REGION Network 1: Conversion de temperatura leida por termopares a temperaturas para poder tratar en el codigo
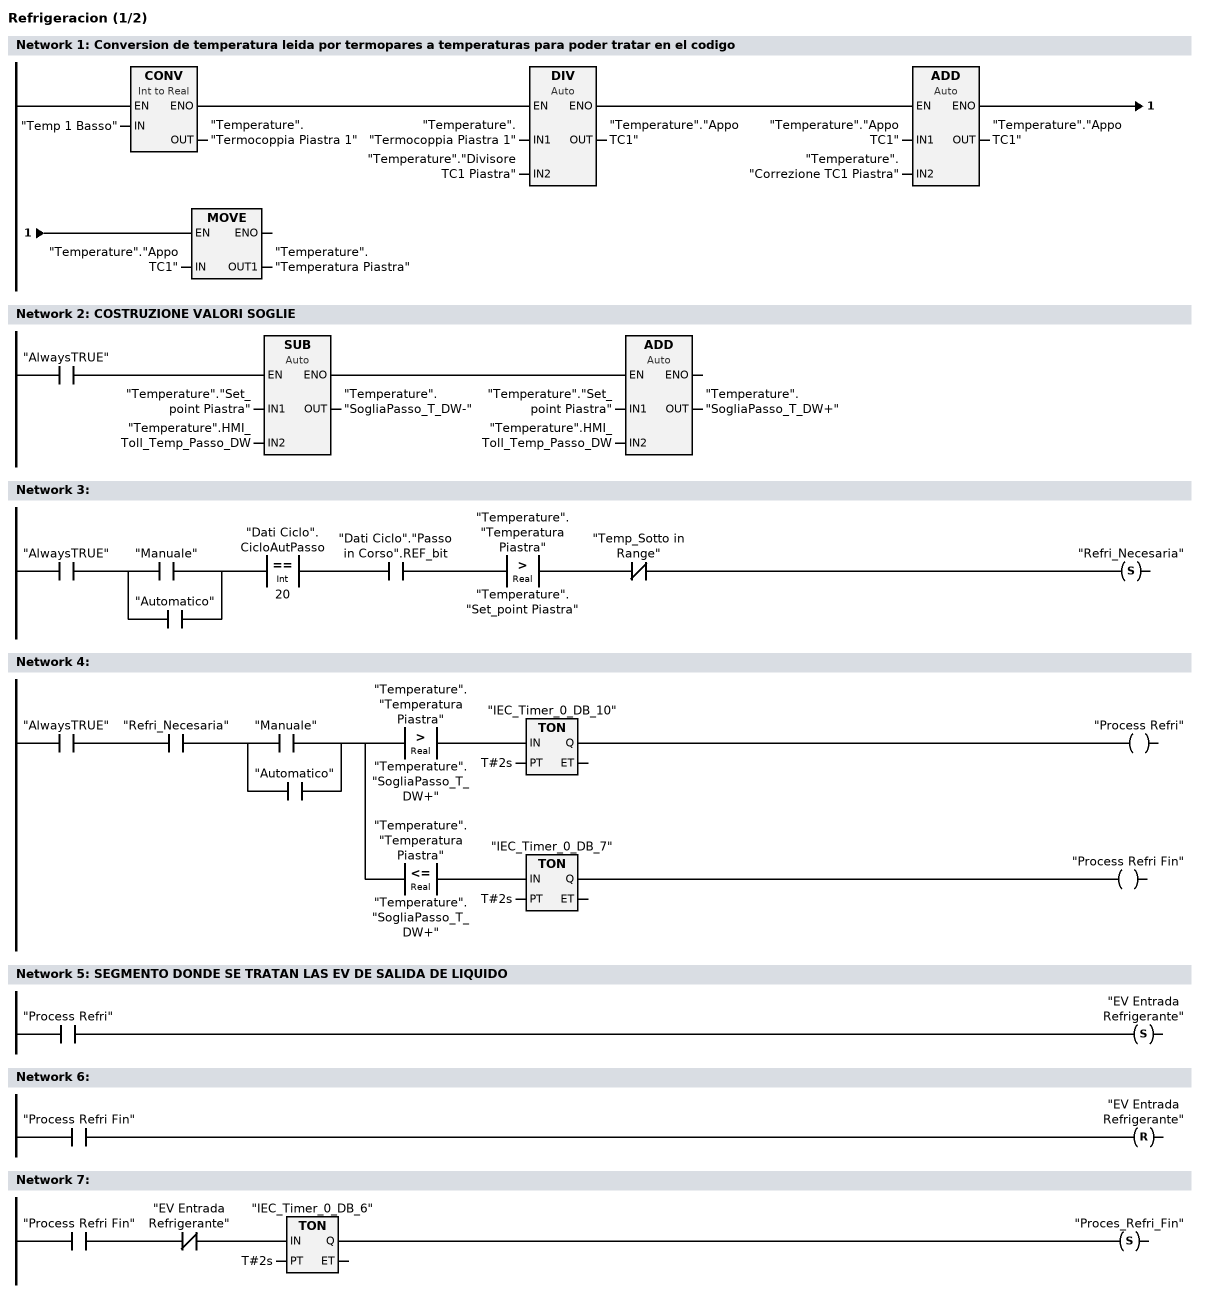
   RUNG wire#powerrail
      { S7_Templates := "[SrcType := Int, DestType := Real]" } Convert(in := "Temp 1 Basso", out => "Temperature"."Termocoppia Piastra 1")
      Div(in1 := "Temperature"."Termocoppia Piastra 1", in2 := "Temperature"."Divisore TC1 Piastra", out => "Temperature"."Appo TC1")
      Add(in1 := "Temperature"."Appo TC1", in2 := "Temperature"."Correzione TC1 Piastra", out => "Temperature"."Appo TC1")
      Move(in := "Temperature"."Appo TC1", out1 => "Temperature"."Temperatura Piastra")
   END_RUNG
   // the same network as SCL:
   "Temperature"."Termocoppia Piastra 1" := INT_TO_REAL("Temp 1 Basso");
   "Temperature"."Appo TC1" := "Temperature"."Termocoppia Piastra 1" / "Temperature"."Divisore TC1 Piastra";
   "Temperature"."Appo TC1" := "Temperature"."Appo TC1" + "Temperature"."Correzione TC1 Piastra";
   "Temperature"."Temperatura Piastra" := "Temperature"."Appo TC1";
END_REGION

REGION Network 2: COSTRUZIONE VALORI SOGLIE
   RUNG wire#powerrail
      Contact( "AlwaysTRUE" )
      Sub(in1 := "Temperature"."Set_point Piastra", in2 := "Temperature".HMI_Toll_Temp_Passo_DW, out => "Temperature"."SogliaPasso_T_DW-")
      Add(in1 := "Temperature"."Set_point Piastra", in2 := "Temperature".HMI_Toll_Temp_Passo_DW, out => "Temperature"."SogliaPasso_T_DW+")
   END_RUNG
   // the same network as SCL:
   IF "AlwaysTRUE" THEN
       "Temperature"."SogliaPasso_T_DW-" := "Temperature"."Set_point Piastra" - "Temperature".HMI_Toll_Temp_Passo_DW;
       "Temperature"."SogliaPasso_T_DW+" := "Temperature"."Set_point Piastra" + "Temperature".HMI_Toll_Temp_Passo_DW;
   END_IF;
END_REGION

REGION Network 3
   RUNG wire#powerrail
      Contact( "AlwaysTRUE" )
      wire#w1
      Contact( "Manuale" )
      wire#w2
      { S7_Templates := "SrcType := Int" } EQ_Contact(in1 := "Dati Ciclo".CicloAutPasso, in2 := 20)
      Contact( "Dati Ciclo"."Passo in Corso".REF_bit )
      { S7_Templates := "SrcType := Real" } GT_Contact(in1 := "Temperature"."Temperatura Piastra", in2 := "Temperature"."Set_point Piastra")
      I_Contact( "Temp_Sotto in Range" )
      S_Coil( "Refri_Necesaria" )
   END_RUNG
   RUNG wire#w1
      Contact( "Automatico" )
   END_RUNG wire#w2
   // the same network as SCL:
   IF "AlwaysTRUE" AND ("Manuale" OR "Automatico") AND ("Dati Ciclo".CicloAutPasso = 20) AND "Dati Ciclo"."Passo in Corso".REF_bit AND ("Temperature"."Temperatura Piastra" > "Temperature"."Set_point Piastra") AND NOT "Temp_Sotto in Range" THEN
       "Refri_Necesaria" := TRUE;
   END_IF;
END_REGION

REGION Network 4
   #_w1 := "AlwaysTRUE" AND "Refri_Necesaria" AND ("Manuale" OR "Automatico");
   "IEC_Timer_0_DB_10".TON(IN := #_w1 AND ("Temperature"."Temperatura Piastra" > "Temperature"."SogliaPasso_T_DW+"),
                           PT := T#2s);
   "Process Refri" := "IEC_Timer_0_DB_10".Q;
   "IEC_Timer_0_DB_7".TON(IN := #_w1 AND ("Temperature"."Temperatura Piastra" <= "Temperature"."SogliaPasso_T_DW+"),
                          PT := T#2s);
   "Process Refri Fin" := "IEC_Timer_0_DB_7".Q;
END_REGION

REGION Network 5: SEGMENTO DONDE SE TRATAN LAS EV DE SALIDA DE LIQUIDO
   RUNG wire#powerrail
      Contact( "Process Refri" )
      S_Coil( "EV Entrada Refrigerante" )
   END_RUNG
   // the same network as SCL:
   IF "Process Refri" THEN "EV Entrada Refrigerante" := TRUE; END_IF;
END_REGION

REGION Network 6
   RUNG wire#powerrail
      Contact( "Process Refri Fin" )
      R_Coil( "EV Entrada Refrigerante" )
   END_RUNG
   // the same network as SCL:
   IF "Process Refri Fin" THEN "EV Entrada Refrigerante" := FALSE; END_IF;
END_REGION

REGION Network 7
   "IEC_Timer_0_DB_6".TON(IN := "Process Refri Fin" AND NOT "EV Entrada Refrigerante", PT := T#2s);
   IF "IEC_Timer_0_DB_6".Q THEN "Proces_Refri_Fin" := TRUE; END_IF;
END_REGION

REGION Network 8
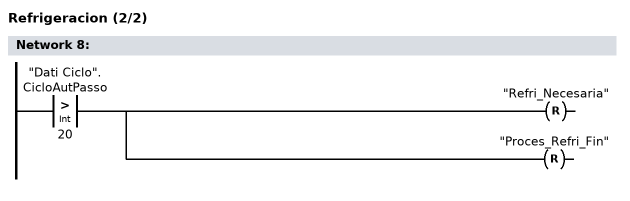
   RUNG wire#powerrail
      { S7_Templates := "SrcType := Int" } GT_Contact(in1 := "Dati Ciclo".CicloAutPasso, in2 := 20)
      wire#w1
      R_Coil( "Refri_Necesaria" )
   END_RUNG
   RUNG wire#w1
      R_Coil( "Proces_Refri_Fin" )
   END_RUNG
   // the same network as SCL:
   IF "Dati Ciclo".CicloAutPasso > 20 THEN
       "Refri_Necesaria" := FALSE;
       "Proces_Refri_Fin" := FALSE;
   END_IF;
END_REGION
END_FUNCTION

FUNCTION "Temperatura Sopra" : Void   // FC11, LAD
{ S7_Optimized_Access := 'TRUE' }
VERSION : 0.1
   VAR_TEMP   // added for the SCL form of the ladder/FBD networks
      _w1 : Bool;
   END_VAR
BEGIN

REGION Network 1: Costruzione valore temperatura
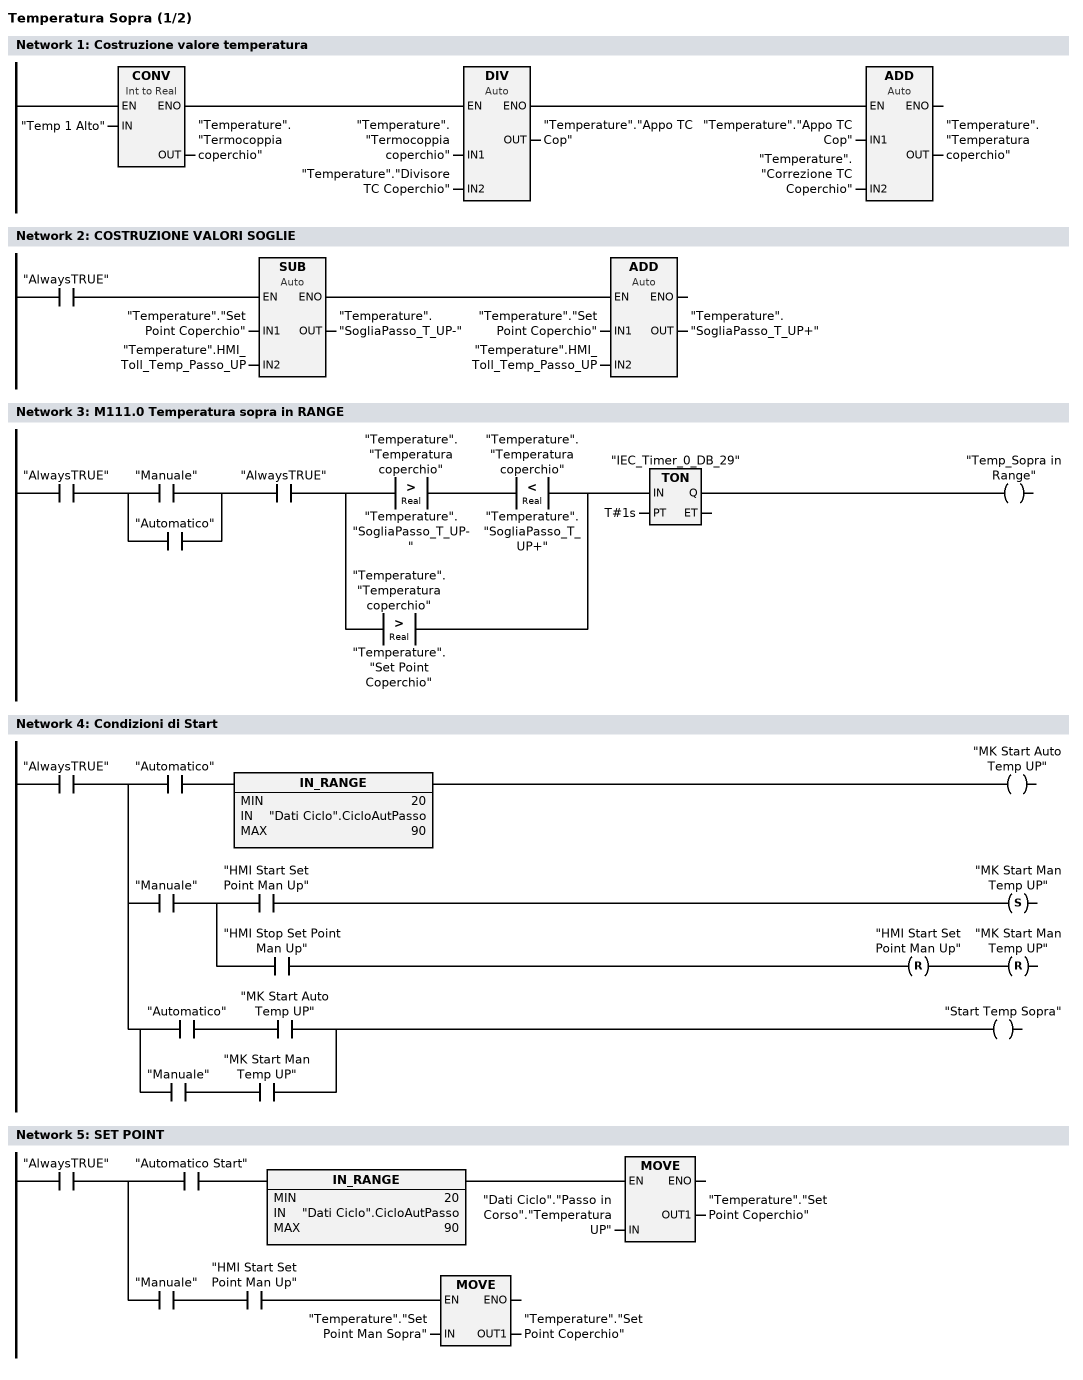
   RUNG wire#powerrail
      { S7_Templates := "[SrcType := Int, DestType := Real]" } Convert(in := "Temp 1 Alto", out => "Temperature"."Termocoppia coperchio")
      Div(in1 := "Temperature"."Termocoppia coperchio", in2 := "Temperature"."Divisore TC Coperchio", out => "Temperature"."Appo TC Cop")
      Add(in1 := "Temperature"."Appo TC Cop", in2 := "Temperature"."Correzione TC Coperchio", out => "Temperature"."Temperatura coperchio")
   END_RUNG
   // the same network as SCL:
   "Temperature"."Termocoppia coperchio" := INT_TO_REAL("Temp 1 Alto");
   "Temperature"."Appo TC Cop" := "Temperature"."Termocoppia coperchio" / "Temperature"."Divisore TC Coperchio";
   "Temperature"."Temperatura coperchio" := "Temperature"."Appo TC Cop" + "Temperature"."Correzione TC Coperchio";
END_REGION

REGION Network 2: COSTRUZIONE VALORI SOGLIE
   RUNG wire#powerrail
      Contact( "AlwaysTRUE" )
      Sub(in1 := "Temperature"."Set Point Coperchio", in2 := "Temperature".HMI_Toll_Temp_Passo_UP, out => "Temperature"."SogliaPasso_T_UP-")
      Add(in1 := "Temperature"."Set Point Coperchio", in2 := "Temperature".HMI_Toll_Temp_Passo_UP, out => "Temperature"."SogliaPasso_T_UP+")
   END_RUNG
   // the same network as SCL:
   IF "AlwaysTRUE" THEN
       "Temperature"."SogliaPasso_T_UP-" := "Temperature"."Set Point Coperchio" - "Temperature".HMI_Toll_Temp_Passo_UP;
       "Temperature"."SogliaPasso_T_UP+" := "Temperature"."Set Point Coperchio" + "Temperature".HMI_Toll_Temp_Passo_UP;
   END_IF;
END_REGION

REGION Network 3: M111.0 Temperatura sopra in RANGE
   "IEC_Timer_0_DB_29".TON(IN := "AlwaysTRUE" AND ("Manuale" OR "Automatico") AND "AlwaysTRUE" AND ((("Temperature"."Temperatura coperchio" > "Temperature"."SogliaPasso_T_UP-") AND ("Temperature"."Temperatura coperchio" < "Temperature"."SogliaPasso_T_UP+")) OR ("Temperature"."Temperatura coperchio" > "Temperature"."Set Point Coperchio")),
                           PT := T#1s);
   "Temp_Sopra in Range" := "IEC_Timer_0_DB_29".Q;
END_REGION

REGION Network 4: Condizioni di Start
   RUNG wire#powerrail
      Contact( "AlwaysTRUE" )
      wire#w1
      Contact( "Automatico" )
      { S7_Templates := "SrcType := Int" } InRange(min := 20, in := "Dati Ciclo".CicloAutPasso, max := 90)
      Coil( "MK Start Auto Temp UP" )
   END_RUNG
   RUNG wire#w1
      Contact( "Manuale" )
      wire#w2
      Contact( "HMI Start Set Point Man Up" )
      S_Coil( "MK Start Man Temp UP" )
   END_RUNG
   RUNG wire#w2
      Contact( "HMI Stop Set Point Man Up" )
      R_Coil( "HMI Start Set Point Man Up" )
      R_Coil( "MK Start Man Temp UP" )
   END_RUNG
   RUNG wire#w1
      Contact( "Automatico" )
      Contact( "MK Start Auto Temp UP" )
      wire#w3
      Coil( "Start Temp Sopra" )
   END_RUNG
   RUNG wire#w1
      Contact( "Manuale" )
      Contact( "MK Start Man Temp UP" )
   END_RUNG wire#w3
   // the same network as SCL:
   "MK Start Auto Temp UP" := "AlwaysTRUE" AND "Automatico" AND (20 <= "Dati Ciclo".CicloAutPasso) AND ("Dati Ciclo".CicloAutPasso <= 90);
   #_w1 := "AlwaysTRUE" AND "Manuale";
   IF #_w1 AND "HMI Start Set Point Man Up" THEN "MK Start Man Temp UP" := TRUE; END_IF;
   IF #_w1 AND "HMI Stop Set Point Man Up" THEN
       "HMI Start Set Point Man Up" := FALSE;
       "MK Start Man Temp UP" := FALSE;
   END_IF;
   "Start Temp Sopra" := "AlwaysTRUE" AND (("Automatico" AND "MK Start Auto Temp UP") OR ("Manuale" AND "MK Start Man Temp UP"));
END_REGION

REGION Network 5: SET POINT
   RUNG wire#powerrail
      Contact( "AlwaysTRUE" )
      wire#w1
      Contact( "Automatico Start" )
      { S7_Templates := "SrcType := Int" } InRange(min := 20, in := "Dati Ciclo".CicloAutPasso, max := 90)
      Move(in := "Dati Ciclo"."Passo in Corso"."Temperatura UP", out1 => "Temperature"."Set Point Coperchio")
   END_RUNG
   RUNG wire#w1
      Contact( "Manuale" )
      Contact( "HMI Start Set Point Man Up" )
      Move(in := "Temperature"."Set Point Man Sopra", out1 => "Temperature"."Set Point Coperchio")
   END_RUNG
   // the same network as SCL:
   IF "AlwaysTRUE" AND "Automatico Start" AND (20 <= "Dati Ciclo".CicloAutPasso) AND ("Dati Ciclo".CicloAutPasso <= 90) THEN
       "Temperature"."Set Point Coperchio" := "Dati Ciclo"."Passo in Corso"."Temperatura UP";
   END_IF;
   IF "AlwaysTRUE" AND "Manuale" AND "HMI Start Set Point Man Up" THEN
       "Temperature"."Set Point Coperchio" := "Temperature"."Set Point Man Sopra";
   END_IF;
END_REGION

REGION Network 6: Comando resistenze
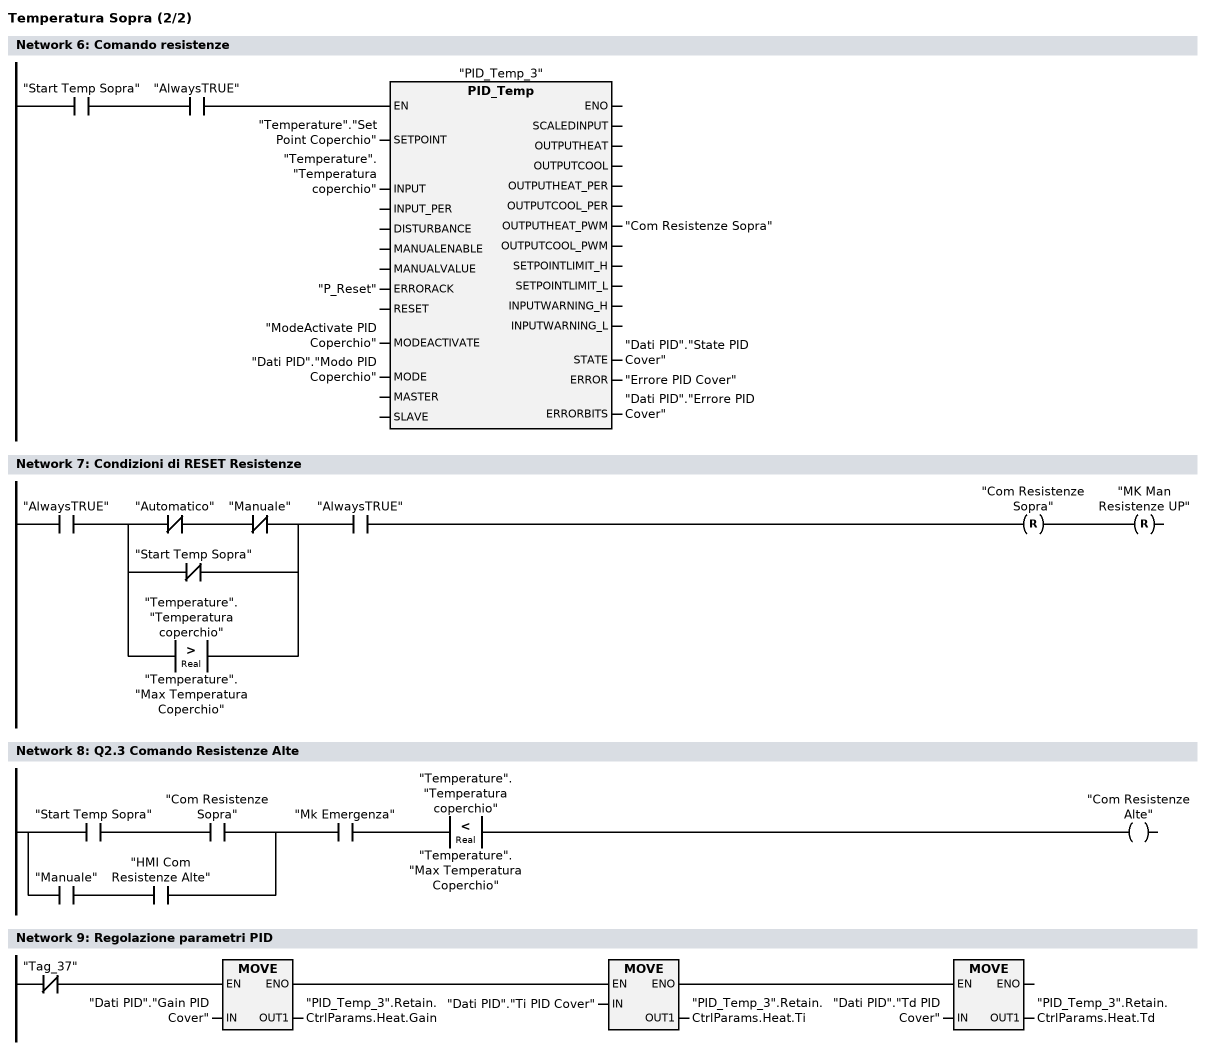
   IF "Start Temp Sopra" AND "AlwaysTRUE" THEN
       "PID_Temp_3"(Setpoint := "Temperature"."Set Point Coperchio",   // PID_Temp
                    Input := "Temperature"."Temperatura coperchio",
                    ErrorAck := "P_Reset",
                    ModeActivate := "ModeActivate PID Coperchio",
                    Mode := "Dati PID"."Modo PID Coperchio",
                    OutputHeat_PWM => "Com Resistenze Sopra",
                    State => "Dati PID"."State PID Cover",
                    Error => "Errore PID Cover",
                    ErrorBits => "Dati PID"."Errore PID Cover");
   END_IF;
END_REGION

REGION Network 7: Condizioni di RESET Resistenze
   RUNG wire#powerrail
      Contact( "AlwaysTRUE" )
      wire#w1
      I_Contact( "Automatico" )
      I_Contact( "Manuale" )
      wire#w2
      Contact( "AlwaysTRUE" )
      R_Coil( "Com Resistenze Sopra" )
      R_Coil( "MK Man Resistenze UP" )
   END_RUNG
   RUNG wire#w1
      I_Contact( "Start Temp Sopra" )
   END_RUNG wire#w2
   RUNG wire#w1
      { S7_Templates := "SrcType := Real" } GT_Contact(in1 := "Temperature"."Temperatura coperchio", in2 := "Temperature"."Max Temperatura Coperchio")
   END_RUNG wire#w2
   // the same network as SCL:
   IF "AlwaysTRUE" AND ((NOT "Automatico" AND NOT "Manuale") OR NOT "Start Temp Sopra" OR ("Temperature"."Temperatura coperchio" > "Temperature"."Max Temperatura Coperchio")) AND "AlwaysTRUE" THEN
       "Com Resistenze Sopra" := FALSE;
       "MK Man Resistenze UP" := FALSE;
   END_IF;
END_REGION

REGION Network 8: Q2.3 Comando Resistenze Alte
   RUNG wire#powerrail
      Contact( "Start Temp Sopra" )
      Contact( "Com Resistenze Sopra" )
      wire#w1
      Contact( "Mk Emergenza" )
      { S7_Templates := "SrcType := Real" } LT_Contact(in1 := "Temperature"."Temperatura coperchio", in2 := "Temperature"."Max Temperatura Coperchio")
      Coil( "Com Resistenze Alte" )
   END_RUNG
   RUNG wire#powerrail
      Contact( "Manuale" )
      Contact( "HMI Com Resistenze Alte" )
   END_RUNG wire#w1
   // the same network as SCL:
   "Com Resistenze Alte" := (("Start Temp Sopra" AND "Com Resistenze Sopra") OR ("Manuale" AND "HMI Com Resistenze Alte")) AND "Mk Emergenza" AND ("Temperature"."Temperatura coperchio" < "Temperature"."Max Temperatura Coperchio");
END_REGION

REGION Network 9: Regolazione parametri PID
   RUNG wire#powerrail
      I_Contact( "Tag_37" )
      Move(in := "Dati PID"."Gain PID Cover", out1 => "PID_Temp_3".Retain.CtrlParams.Heat.Gain)
      Move(in := "Dati PID"."Ti PID Cover", out1 => "PID_Temp_3".Retain.CtrlParams.Heat.Ti)
      Move(in := "Dati PID"."Td PID Cover", out1 => "PID_Temp_3".Retain.CtrlParams.Heat.Td)
   END_RUNG
   // the same network as SCL:
   IF NOT "Tag_37" THEN
       "PID_Temp_3".Retain.CtrlParams.Heat.Gain := "Dati PID"."Gain PID Cover";
       "PID_Temp_3".Retain.CtrlParams.Heat.Ti := "Dati PID"."Ti PID Cover";
       "PID_Temp_3".Retain.CtrlParams.Heat.Td := "Dati PID"."Td PID Cover";
   END_IF;
END_REGION
END_FUNCTION

FUNCTION "Vuoto Sotto" : Void   // FC12, LAD
{ S7_Optimized_Access := 'TRUE' }
VERSION : 0.1
   VAR_TEMP   // added for the SCL form of the ladder/FBD networks
      _w1 : Bool;
      _w2 : Bool;
   END_VAR
BEGIN

REGION Network 1: Costruzione valore vuoto
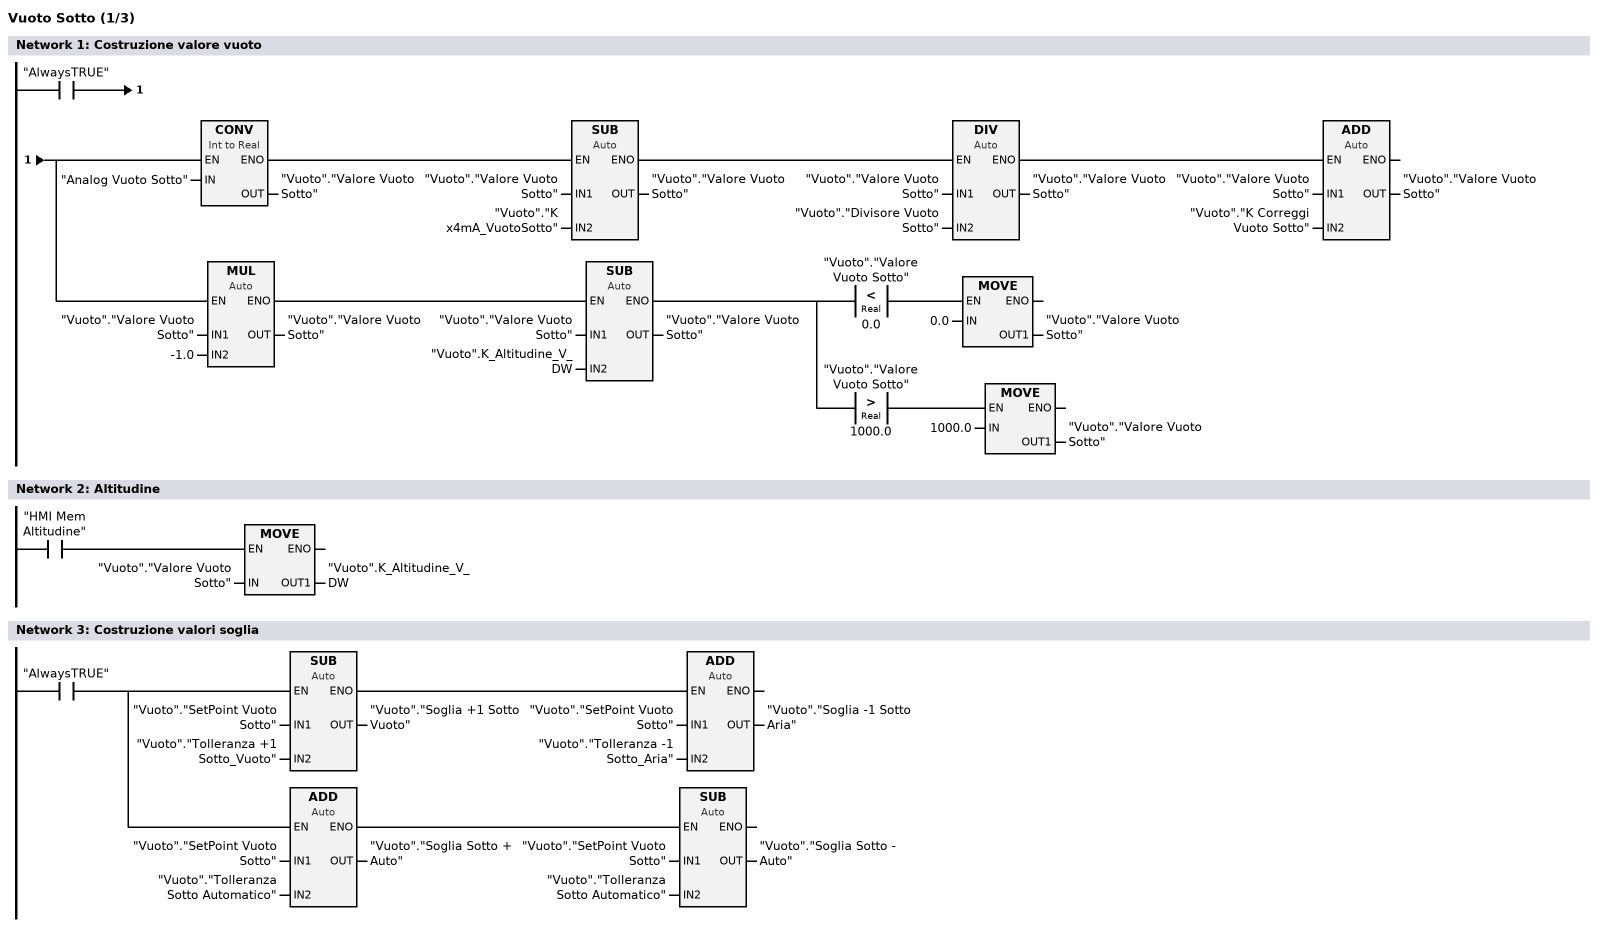
   RUNG wire#powerrail
      Contact( "AlwaysTRUE" )
      wire#w1
      { S7_Templates := "[SrcType := Int, DestType := Real]" } Convert(in := "Analog Vuoto Sotto", out => "Vuoto"."Valore Vuoto Sotto")
      Sub(in1 := "Vuoto"."Valore Vuoto Sotto", in2 := "Vuoto"."K x4mA_VuotoSotto", out => "Vuoto"."Valore Vuoto Sotto")
      Div(in1 := "Vuoto"."Valore Vuoto Sotto", in2 := "Vuoto"."Divisore Vuoto Sotto", out => "Vuoto"."Valore Vuoto Sotto")
      Add(in1 := "Vuoto"."Valore Vuoto Sotto", in2 := "Vuoto"."K Correggi Vuoto Sotto", out => "Vuoto"."Valore Vuoto Sotto")
   END_RUNG
   RUNG wire#w1
      Mul(in1 := "Vuoto"."Valore Vuoto Sotto", in2 := -1.0, out => "Vuoto"."Valore Vuoto Sotto")
      Sub(in1 := "Vuoto"."Valore Vuoto Sotto", in2 := "Vuoto".K_Altitudine_V_DW, out => "Vuoto"."Valore Vuoto Sotto")
      wire#w2
      { S7_Templates := "SrcType := Real" } LT_Contact(in1 := "Vuoto"."Valore Vuoto Sotto", in2 := 0.0)
      Move(in := 0.0, out1 => "Vuoto"."Valore Vuoto Sotto")
   END_RUNG
   RUNG wire#w2
      { S7_Templates := "SrcType := Real" } GT_Contact(in1 := "Vuoto"."Valore Vuoto Sotto", in2 := 1000.0)
      Move(in := 1000.0, out1 => "Vuoto"."Valore Vuoto Sotto")
   END_RUNG
   // the same network as SCL:
   IF "AlwaysTRUE" THEN
       "Vuoto"."Valore Vuoto Sotto" := INT_TO_REAL("Analog Vuoto Sotto");
       "Vuoto"."Valore Vuoto Sotto" := "Vuoto"."Valore Vuoto Sotto" - "Vuoto"."K x4mA_VuotoSotto";
       "Vuoto"."Valore Vuoto Sotto" := "Vuoto"."Valore Vuoto Sotto" / "Vuoto"."Divisore Vuoto Sotto";
       "Vuoto"."Valore Vuoto Sotto" := "Vuoto"."Valore Vuoto Sotto" + "Vuoto"."K Correggi Vuoto Sotto";
       "Vuoto"."Valore Vuoto Sotto" := "Vuoto"."Valore Vuoto Sotto" * (-1.0);
       "Vuoto"."Valore Vuoto Sotto" := "Vuoto"."Valore Vuoto Sotto" - "Vuoto".K_Altitudine_V_DW;
   END_IF;
   IF "AlwaysTRUE" AND ("Vuoto"."Valore Vuoto Sotto" < 0.0) THEN "Vuoto"."Valore Vuoto Sotto" := 0.0; END_IF;
   IF "AlwaysTRUE" AND ("Vuoto"."Valore Vuoto Sotto" > 1000.0) THEN
       "Vuoto"."Valore Vuoto Sotto" := 1000.0;
   END_IF;
END_REGION

REGION Network 2: Altitudine
   RUNG wire#powerrail
      Contact( "HMI Mem Altitudine" )
      Move(in := "Vuoto"."Valore Vuoto Sotto", out1 => "Vuoto".K_Altitudine_V_DW)
   END_RUNG
   // the same network as SCL:
   IF "HMI Mem Altitudine" THEN "Vuoto".K_Altitudine_V_DW := "Vuoto"."Valore Vuoto Sotto"; END_IF;
END_REGION

REGION Network 3: Costruzione valori soglia
   RUNG wire#powerrail
      Contact( "AlwaysTRUE" )
      wire#w1
      Sub(in1 := "Vuoto"."SetPoint Vuoto Sotto", in2 := "Vuoto"."Tolleranza +1 Sotto_Vuoto", out => "Vuoto"."Soglia +1 Sotto Vuoto")
      Add(in1 := "Vuoto"."SetPoint Vuoto Sotto", in2 := "Vuoto"."Tolleranza -1 Sotto_Aria", out => "Vuoto"."Soglia -1 Sotto Aria")
   END_RUNG
   RUNG wire#w1
      Add(in1 := "Vuoto"."SetPoint Vuoto Sotto", in2 := "Vuoto"."Tolleranza Sotto Automatico", out => "Vuoto"."Soglia Sotto + Auto")
      Sub(in1 := "Vuoto"."SetPoint Vuoto Sotto", in2 := "Vuoto"."Tolleranza Sotto Automatico", out => "Vuoto"."Soglia Sotto - Auto")
   END_RUNG
   // the same network as SCL:
   IF "AlwaysTRUE" THEN
       "Vuoto"."Soglia +1 Sotto Vuoto" := "Vuoto"."SetPoint Vuoto Sotto" - "Vuoto"."Tolleranza +1 Sotto_Vuoto";
       "Vuoto"."Soglia -1 Sotto Aria" := "Vuoto"."SetPoint Vuoto Sotto" + "Vuoto"."Tolleranza -1 Sotto_Aria";
       "Vuoto"."Soglia Sotto + Auto" := "Vuoto"."SetPoint Vuoto Sotto" + "Vuoto"."Tolleranza Sotto Automatico";
       "Vuoto"."Soglia Sotto - Auto" := "Vuoto"."SetPoint Vuoto Sotto" - "Vuoto"."Tolleranza Sotto Automatico";
   END_IF;
END_REGION

REGION Network 4: Condizioni di start
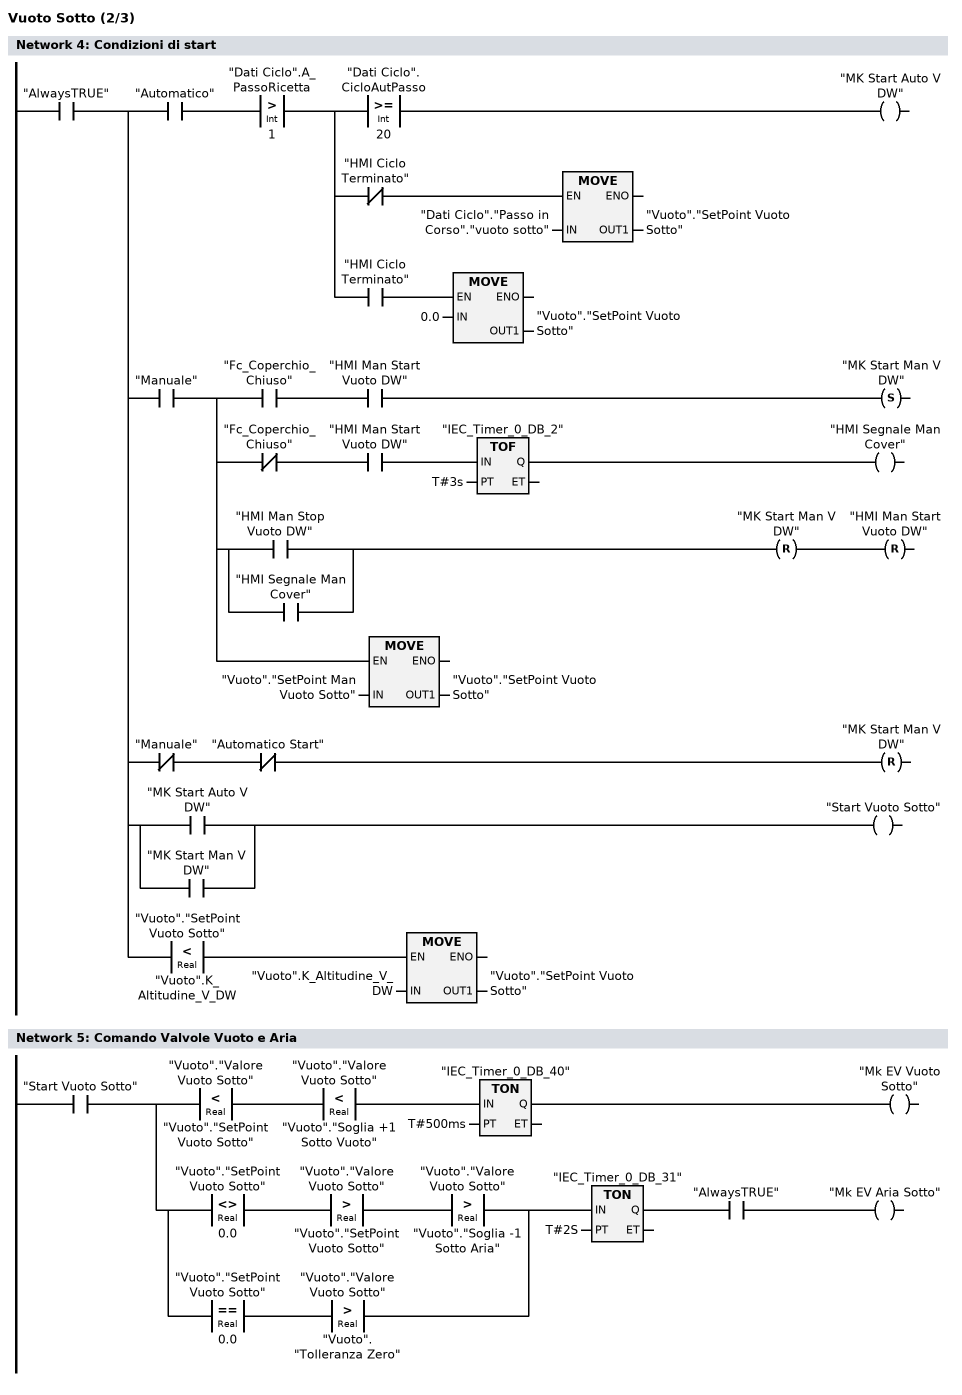
   #_w1 := "AlwaysTRUE" AND "Automatico" AND ("Dati Ciclo".A_PassoRicetta > 1);
   "MK Start Auto V DW" := #_w1 AND ("Dati Ciclo".CicloAutPasso >= 20);
   IF #_w1 AND NOT "HMI Ciclo Terminato" THEN
       "Vuoto"."SetPoint Vuoto Sotto" := "Dati Ciclo"."Passo in Corso"."vuoto sotto";
   END_IF;
   IF #_w1 AND "HMI Ciclo Terminato" THEN "Vuoto"."SetPoint Vuoto Sotto" := 0.0; END_IF;
   #_w2 := "AlwaysTRUE" AND "Manuale";
   IF #_w2 AND "Fc_Coperchio_Chiuso" AND "HMI Man Start Vuoto DW" THEN "MK Start Man V DW" := TRUE; END_IF;
   "IEC_Timer_0_DB_2".TOF(IN := #_w2 AND NOT "Fc_Coperchio_Chiuso" AND "HMI Man Start Vuoto DW", PT := T#3s);
   "HMI Segnale Man Cover" := "IEC_Timer_0_DB_2".Q;
   IF #_w2 AND ("HMI Man Stop Vuoto DW" OR "HMI Segnale Man Cover") THEN
       "MK Start Man V DW" := FALSE;
       "HMI Man Start Vuoto DW" := FALSE;
   END_IF;
   IF #_w2 THEN "Vuoto"."SetPoint Vuoto Sotto" := "Vuoto"."SetPoint Man Vuoto Sotto"; END_IF;
   IF "AlwaysTRUE" AND NOT "Manuale" AND NOT "Automatico Start" THEN "MK Start Man V DW" := FALSE; END_IF;
   "Start Vuoto Sotto" := "AlwaysTRUE" AND ("MK Start Auto V DW" OR "MK Start Man V DW");
   IF "AlwaysTRUE" AND ("Vuoto"."SetPoint Vuoto Sotto" < "Vuoto".K_Altitudine_V_DW) THEN
       "Vuoto"."SetPoint Vuoto Sotto" := "Vuoto".K_Altitudine_V_DW;
   END_IF;
END_REGION

REGION Network 5: Comando Valvole Vuoto e Aria
   "IEC_Timer_0_DB_40".TON(IN := "Start Vuoto Sotto" AND ("Vuoto"."Valore Vuoto Sotto" < "Vuoto"."SetPoint Vuoto Sotto") AND ("Vuoto"."Valore Vuoto Sotto" < "Vuoto"."Soglia +1 Sotto Vuoto"),
                           PT := T#500ms);
   "Mk EV Vuoto Sotto" := "IEC_Timer_0_DB_40".Q;
   "IEC_Timer_0_DB_31".TON(IN := "Start Vuoto Sotto" AND ((("Vuoto"."SetPoint Vuoto Sotto" <> 0.0) AND ("Vuoto"."Valore Vuoto Sotto" > "Vuoto"."SetPoint Vuoto Sotto") AND ("Vuoto"."Valore Vuoto Sotto" > "Vuoto"."Soglia -1 Sotto Aria")) OR (("Vuoto"."SetPoint Vuoto Sotto" = 0.0) AND ("Vuoto"."Valore Vuoto Sotto" > "Vuoto"."Tolleranza Zero"))),
                           PT := T#2S);
   "Mk EV Aria Sotto" := "IEC_Timer_0_DB_31".Q AND "AlwaysTRUE";
END_REGION

REGION Network 6: Vuoto in Range
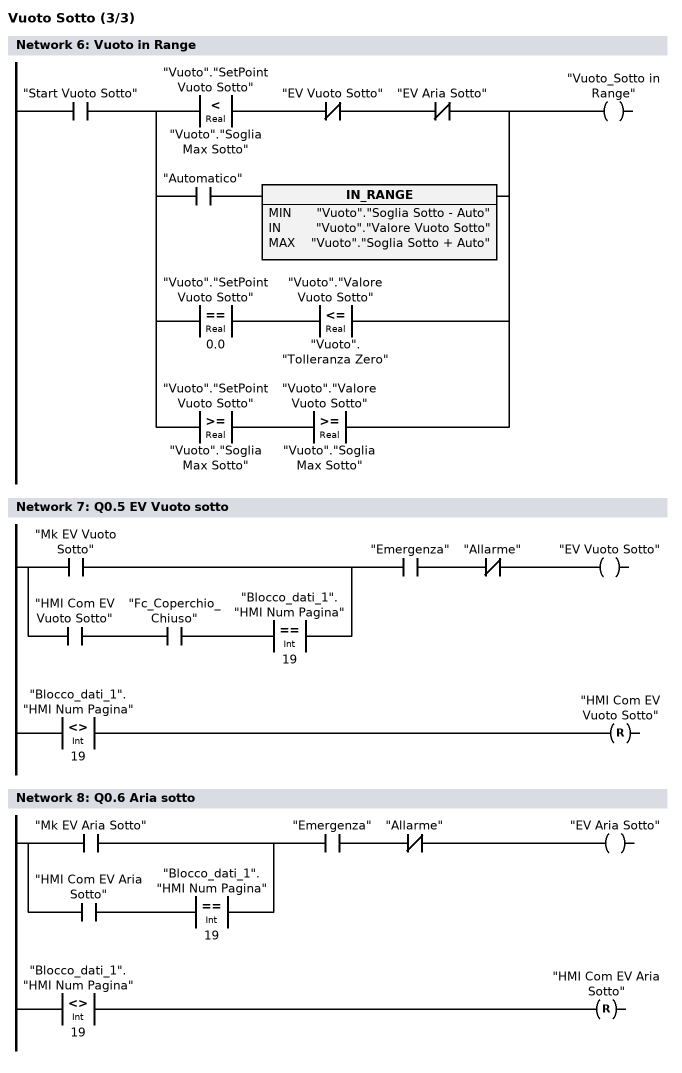
   RUNG wire#powerrail
      Contact( "Start Vuoto Sotto" )
      wire#w1
      { S7_Templates := "SrcType := Real" } LT_Contact(in1 := "Vuoto"."SetPoint Vuoto Sotto", in2 := "Vuoto"."Soglia Max Sotto")
      I_Contact( "EV Vuoto Sotto" )
      I_Contact( "EV Aria Sotto" )
      wire#w2
      Coil( "Vuoto_Sotto in Range" )
   END_RUNG
   RUNG wire#w1
      Contact( "Automatico" )
      { S7_Templates := "SrcType := Real" } InRange(min := "Vuoto"."Soglia Sotto - Auto", in := "Vuoto"."Valore Vuoto Sotto", max := "Vuoto"."Soglia Sotto + Auto")
   END_RUNG wire#w2
   RUNG wire#w1
      { S7_Templates := "SrcType := Real" } EQ_Contact(in1 := "Vuoto"."SetPoint Vuoto Sotto", in2 := 0.0)
      { S7_Templates := "SrcType := Real" } LE_Contact(in1 := "Vuoto"."Valore Vuoto Sotto", in2 := "Vuoto"."Tolleranza Zero")
   END_RUNG wire#w2
   RUNG wire#w1
      { S7_Templates := "SrcType := Real" } GE_Contact(in1 := "Vuoto"."SetPoint Vuoto Sotto", in2 := "Vuoto"."Soglia Max Sotto")
      { S7_Templates := "SrcType := Real" } GE_Contact(in1 := "Vuoto"."Valore Vuoto Sotto", in2 := "Vuoto"."Soglia Max Sotto")
   END_RUNG wire#w2
   // the same network as SCL:
   "Vuoto_Sotto in Range" := "Start Vuoto Sotto" AND ((("Vuoto"."SetPoint Vuoto Sotto" < "Vuoto"."Soglia Max Sotto") AND NOT "EV Vuoto Sotto" AND NOT "EV Aria Sotto") OR ("Automatico" AND ("Vuoto"."Soglia Sotto - Auto" <= "Vuoto"."Valore Vuoto Sotto") AND ("Vuoto"."Valore Vuoto Sotto" <= "Vuoto"."Soglia Sotto + Auto")) OR (("Vuoto"."SetPoint Vuoto Sotto" = 0.0) AND ("Vuoto"."Valore Vuoto Sotto" <= "Vuoto"."Tolleranza Zero")) OR (("Vuoto"."SetPoint Vuoto Sotto" >= "Vuoto"."Soglia Max Sotto") AND ("Vuoto"."Valore Vuoto Sotto" >= "Vuoto"."Soglia Max Sotto")));
END_REGION

REGION Network 7: Q0.5 EV Vuoto sotto
   RUNG wire#powerrail
      Contact( "Mk EV Vuoto Sotto" )
      wire#w1
      Contact( "Emergenza" )
      I_Contact( "Allarme" )
      Coil( "EV Vuoto Sotto" )
   END_RUNG
   RUNG wire#powerrail
      Contact( "HMI Com EV Vuoto Sotto" )
      Contact( "Fc_Coperchio_Chiuso" )
      { S7_Templates := "SrcType := Int" } EQ_Contact(in1 := "Blocco_dati_1"."HMI Num Pagina", in2 := 19)
   END_RUNG wire#w1
   RUNG wire#powerrail
      { S7_Templates := "SrcType := Int" } NE_Contact(in1 := "Blocco_dati_1"."HMI Num Pagina", in2 := 19)
      R_Coil( "HMI Com EV Vuoto Sotto" )
   END_RUNG
   // the same network as SCL:
   "EV Vuoto Sotto" := ("Mk EV Vuoto Sotto" OR ("HMI Com EV Vuoto Sotto" AND "Fc_Coperchio_Chiuso" AND ("Blocco_dati_1"."HMI Num Pagina" = 19))) AND "Emergenza" AND NOT "Allarme";
   IF "Blocco_dati_1"."HMI Num Pagina" <> 19 THEN "HMI Com EV Vuoto Sotto" := FALSE; END_IF;
END_REGION

REGION Network 8: Q0.6 Aria sotto
   RUNG wire#powerrail
      Contact( "Mk EV Aria Sotto" )
      wire#w1
      Contact( "Emergenza" )
      I_Contact( "Allarme" )
      Coil( "EV Aria Sotto" )
   END_RUNG
   RUNG wire#powerrail
      Contact( "HMI Com EV Aria Sotto" )
      { S7_Templates := "SrcType := Int" } EQ_Contact(in1 := "Blocco_dati_1"."HMI Num Pagina", in2 := 19)
   END_RUNG wire#w1
   RUNG wire#powerrail
      { S7_Templates := "SrcType := Int" } NE_Contact(in1 := "Blocco_dati_1"."HMI Num Pagina", in2 := 19)
      R_Coil( "HMI Com EV Aria Sotto" )
   END_RUNG
   // the same network as SCL:
   "EV Aria Sotto" := ("Mk EV Aria Sotto" OR ("HMI Com EV Aria Sotto" AND ("Blocco_dati_1"."HMI Num Pagina" = 19))) AND "Emergenza" AND NOT "Allarme";
   IF "Blocco_dati_1"."HMI Num Pagina" <> 19 THEN "HMI Com EV Aria Sotto" := FALSE; END_IF;
END_REGION
END_FUNCTION

FUNCTION "Vuoto Sopra" : Void   // FC13, LAD
{ S7_Optimized_Access := 'TRUE' }
VERSION : 0.1
   VAR_TEMP   // added for the SCL form of the ladder/FBD networks
      _w1 : Bool;
      _w2 : Bool;
   END_VAR
BEGIN

REGION Network 1: Costruzione valore vuoto
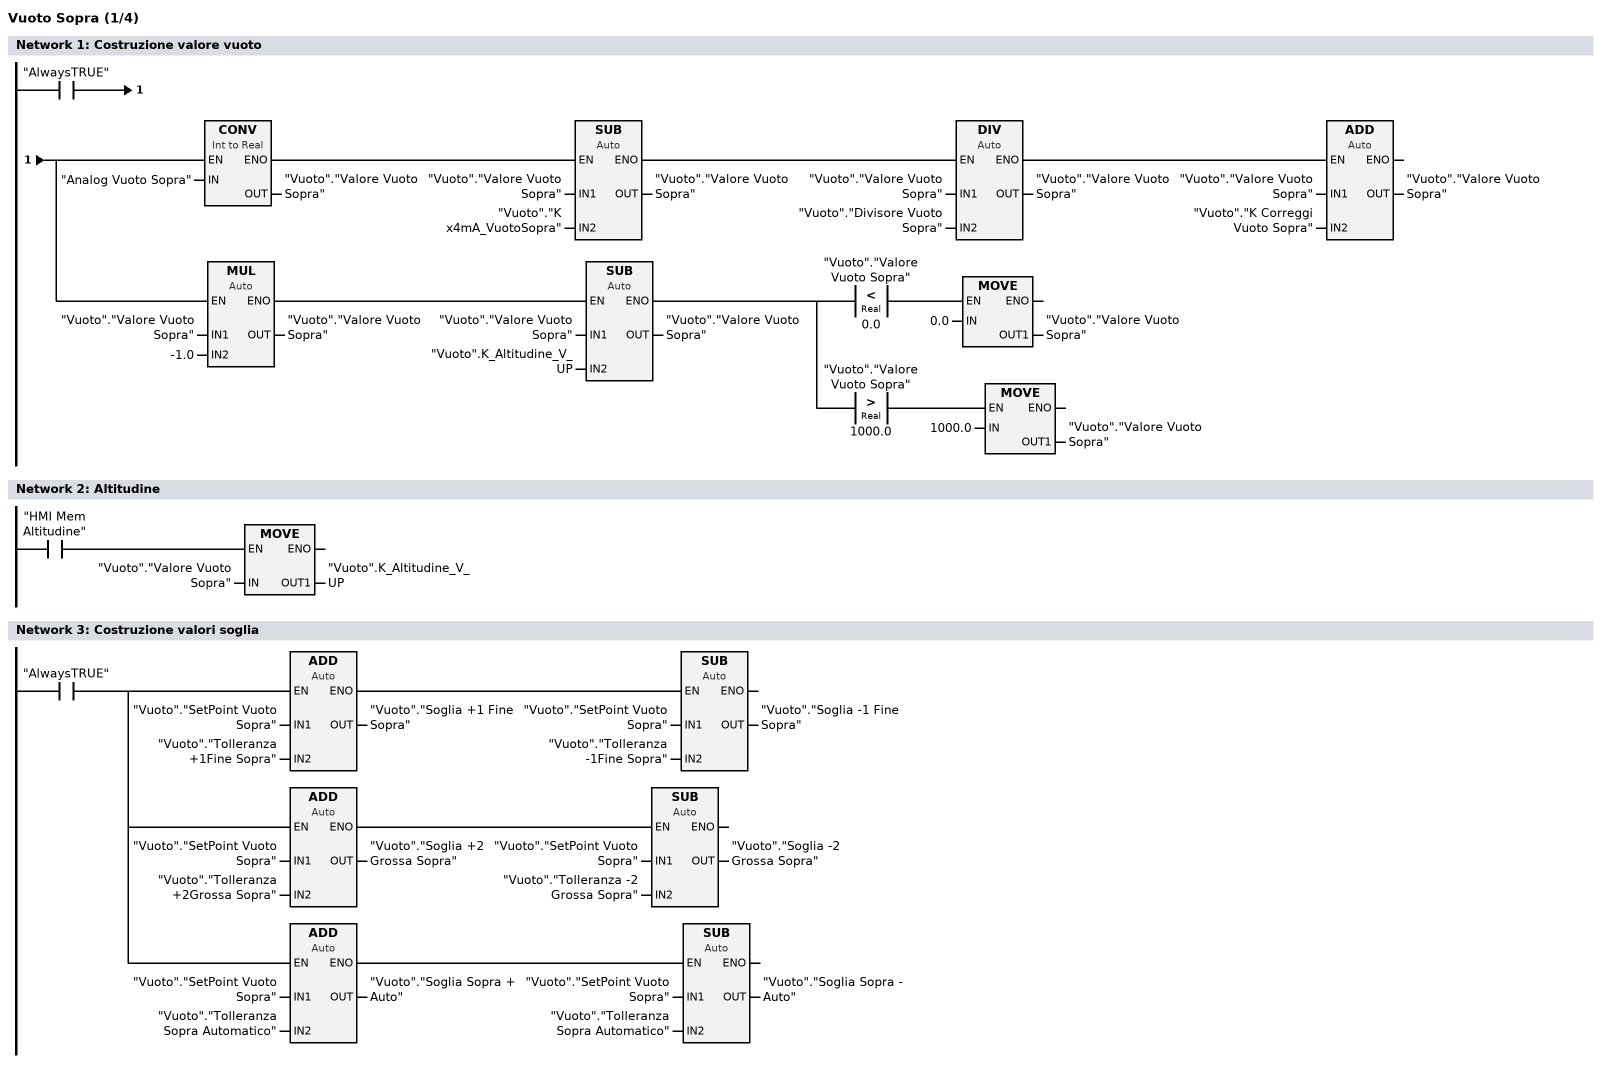
   RUNG wire#powerrail
      Contact( "AlwaysTRUE" )
      wire#w1
      { S7_Templates := "[SrcType := Int, DestType := Real]" } Convert(in := "Analog Vuoto Sopra", out => "Vuoto"."Valore Vuoto Sopra")
      Sub(in1 := "Vuoto"."Valore Vuoto Sopra", in2 := "Vuoto"."K x4mA_VuotoSopra", out => "Vuoto"."Valore Vuoto Sopra")
      Div(in1 := "Vuoto"."Valore Vuoto Sopra", in2 := "Vuoto"."Divisore Vuoto Sopra", out => "Vuoto"."Valore Vuoto Sopra")
      Add(in1 := "Vuoto"."Valore Vuoto Sopra", in2 := "Vuoto"."K Correggi Vuoto Sopra", out => "Vuoto"."Valore Vuoto Sopra")
   END_RUNG
   RUNG wire#w1
      Mul(in1 := "Vuoto"."Valore Vuoto Sopra", in2 := -1.0, out => "Vuoto"."Valore Vuoto Sopra")
      Sub(in1 := "Vuoto"."Valore Vuoto Sopra", in2 := "Vuoto".K_Altitudine_V_UP, out => "Vuoto"."Valore Vuoto Sopra")
      wire#w2
      { S7_Templates := "SrcType := Real" } LT_Contact(in1 := "Vuoto"."Valore Vuoto Sopra", in2 := 0.0)
      Move(in := 0.0, out1 => "Vuoto"."Valore Vuoto Sopra")
   END_RUNG
   RUNG wire#w2
      { S7_Templates := "SrcType := Real" } GT_Contact(in1 := "Vuoto"."Valore Vuoto Sopra", in2 := 1000.0)
      Move(in := 1000.0, out1 => "Vuoto"."Valore Vuoto Sopra")
   END_RUNG
   // the same network as SCL:
   IF "AlwaysTRUE" THEN
       "Vuoto"."Valore Vuoto Sopra" := INT_TO_REAL("Analog Vuoto Sopra");
       "Vuoto"."Valore Vuoto Sopra" := "Vuoto"."Valore Vuoto Sopra" - "Vuoto"."K x4mA_VuotoSopra";
       "Vuoto"."Valore Vuoto Sopra" := "Vuoto"."Valore Vuoto Sopra" / "Vuoto"."Divisore Vuoto Sopra";
       "Vuoto"."Valore Vuoto Sopra" := "Vuoto"."Valore Vuoto Sopra" + "Vuoto"."K Correggi Vuoto Sopra";
       "Vuoto"."Valore Vuoto Sopra" := "Vuoto"."Valore Vuoto Sopra" * (-1.0);
       "Vuoto"."Valore Vuoto Sopra" := "Vuoto"."Valore Vuoto Sopra" - "Vuoto".K_Altitudine_V_UP;
   END_IF;
   IF "AlwaysTRUE" AND ("Vuoto"."Valore Vuoto Sopra" < 0.0) THEN "Vuoto"."Valore Vuoto Sopra" := 0.0; END_IF;
   IF "AlwaysTRUE" AND ("Vuoto"."Valore Vuoto Sopra" > 1000.0) THEN
       "Vuoto"."Valore Vuoto Sopra" := 1000.0;
   END_IF;
END_REGION

REGION Network 2: Altitudine
   RUNG wire#powerrail
      Contact( "HMI Mem Altitudine" )
      Move(in := "Vuoto"."Valore Vuoto Sopra", out1 => "Vuoto".K_Altitudine_V_UP)
   END_RUNG
   // the same network as SCL:
   IF "HMI Mem Altitudine" THEN "Vuoto".K_Altitudine_V_UP := "Vuoto"."Valore Vuoto Sopra"; END_IF;
END_REGION

REGION Network 3: Costruzione valori soglia
   RUNG wire#powerrail
      Contact( "AlwaysTRUE" )
      wire#w1
      Add(in1 := "Vuoto"."SetPoint Vuoto Sopra", in2 := "Vuoto"."Tolleranza +1Fine Sopra", out => "Vuoto"."Soglia +1 Fine Sopra")
      Sub(in1 := "Vuoto"."SetPoint Vuoto Sopra", in2 := "Vuoto"."Tolleranza -1Fine Sopra", out => "Vuoto"."Soglia -1 Fine Sopra")
   END_RUNG
   RUNG wire#w1
      Add(in1 := "Vuoto"."SetPoint Vuoto Sopra", in2 := "Vuoto"."Tolleranza +2Grossa Sopra", out => "Vuoto"."Soglia +2 Grossa Sopra")
      Sub(in1 := "Vuoto"."SetPoint Vuoto Sopra", in2 := "Vuoto"."Tolleranza -2 Grossa Sopra", out => "Vuoto"."Soglia -2 Grossa Sopra")
   END_RUNG
   RUNG wire#w1
      Add(in1 := "Vuoto"."SetPoint Vuoto Sopra", in2 := "Vuoto"."Tolleranza Sopra Automatico", out => "Vuoto"."Soglia Sopra + Auto")
      Sub(in1 := "Vuoto"."SetPoint Vuoto Sopra", in2 := "Vuoto"."Tolleranza Sopra Automatico", out => "Vuoto"."Soglia Sopra - Auto")
   END_RUNG
   // the same network as SCL:
   IF "AlwaysTRUE" THEN
       "Vuoto"."Soglia +1 Fine Sopra" := "Vuoto"."SetPoint Vuoto Sopra" + "Vuoto"."Tolleranza +1Fine Sopra";
       "Vuoto"."Soglia -1 Fine Sopra" := "Vuoto"."SetPoint Vuoto Sopra" - "Vuoto"."Tolleranza -1Fine Sopra";
       "Vuoto"."Soglia +2 Grossa Sopra" := "Vuoto"."SetPoint Vuoto Sopra" + "Vuoto"."Tolleranza +2Grossa Sopra";
       "Vuoto"."Soglia -2 Grossa Sopra" := "Vuoto"."SetPoint Vuoto Sopra" - "Vuoto"."Tolleranza -2 Grossa Sopra";
       "Vuoto"."Soglia Sopra + Auto" := "Vuoto"."SetPoint Vuoto Sopra" + "Vuoto"."Tolleranza Sopra Automatico";
       "Vuoto"."Soglia Sopra - Auto" := "Vuoto"."SetPoint Vuoto Sopra" - "Vuoto"."Tolleranza Sopra Automatico";
   END_IF;
END_REGION

REGION Network 4: Condizioni di start
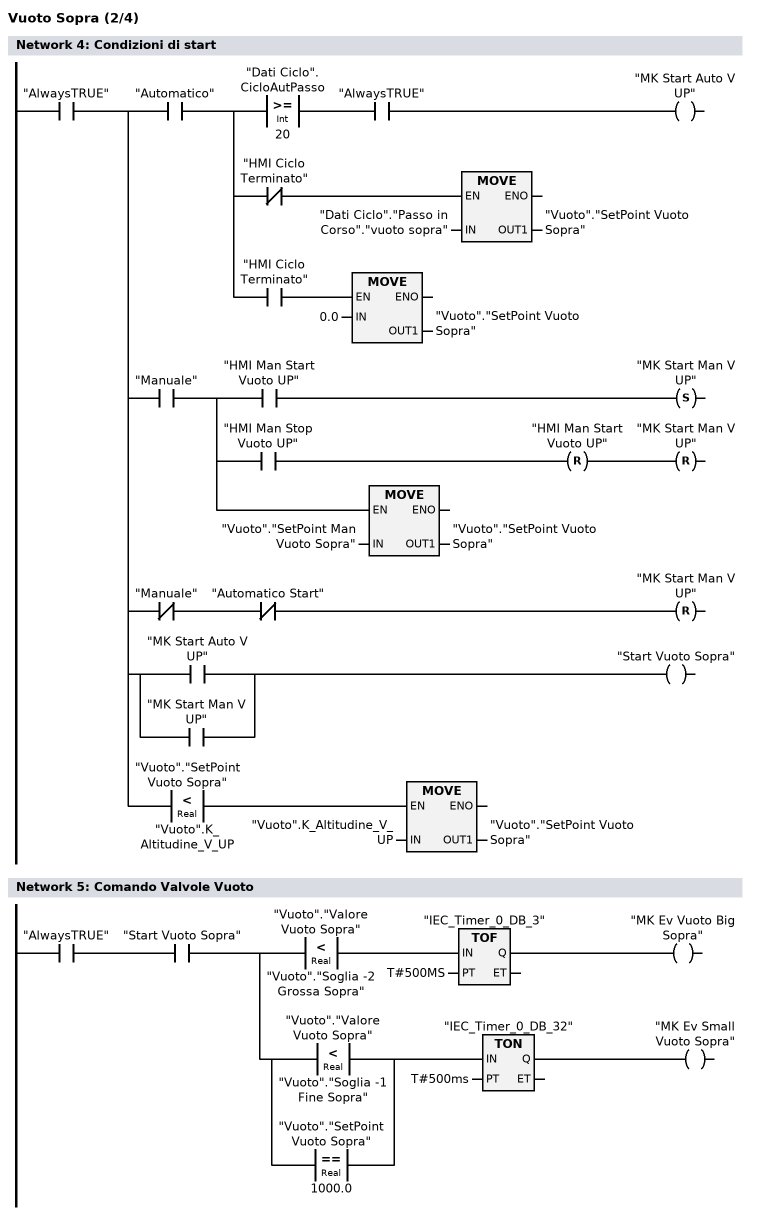
   RUNG wire#powerrail
      Contact( "AlwaysTRUE" )
      wire#w1
      Contact( "Automatico" )
      wire#w2
      { S7_Templates := "SrcType := Int" } GE_Contact(in1 := "Dati Ciclo".CicloAutPasso, in2 := 20)
      Contact( "AlwaysTRUE" )
      Coil( "MK Start Auto V UP" )
   END_RUNG
   RUNG wire#w2
      I_Contact( "HMI Ciclo Terminato" )
      Move(in := "Dati Ciclo"."Passo in Corso"."vuoto sopra", out1 => "Vuoto"."SetPoint Vuoto Sopra")
   END_RUNG
   RUNG wire#w2
      Contact( "HMI Ciclo Terminato" )
      Move(in := 0.0, out1 => "Vuoto"."SetPoint Vuoto Sopra")
   END_RUNG
   RUNG wire#w1
      Contact( "Manuale" )
      wire#w3
      Contact( "HMI Man Start Vuoto UP" )
      S_Coil( "MK Start Man V UP" )
   END_RUNG
   RUNG wire#w3
      Contact( "HMI Man Stop Vuoto UP" )
      R_Coil( "HMI Man Start Vuoto UP" )
      R_Coil( "MK Start Man V UP" )
   END_RUNG
   RUNG wire#w3
      Move(in := "Vuoto"."SetPoint Man Vuoto Sopra", out1 => "Vuoto"."SetPoint Vuoto Sopra")
   END_RUNG
   RUNG wire#w1
      I_Contact( "Manuale" )
      I_Contact( "Automatico Start" )
      R_Coil( "MK Start Man V UP" )
   END_RUNG
   RUNG wire#w1
      Contact( "MK Start Auto V UP" )
      wire#w4
      Coil( "Start Vuoto Sopra" )
   END_RUNG
   RUNG wire#w1
      Contact( "MK Start Man V UP" )
   END_RUNG wire#w4
   RUNG wire#w1
      { S7_Templates := "SrcType := Real" } LT_Contact(in1 := "Vuoto"."SetPoint Vuoto Sopra", in2 := "Vuoto".K_Altitudine_V_UP)
      Move(in := "Vuoto".K_Altitudine_V_UP, out1 => "Vuoto"."SetPoint Vuoto Sopra")
   END_RUNG
   // the same network as SCL:
   #_w1 := "AlwaysTRUE" AND "Automatico";
   "MK Start Auto V UP" := #_w1 AND ("Dati Ciclo".CicloAutPasso >= 20) AND "AlwaysTRUE";
   IF #_w1 AND NOT "HMI Ciclo Terminato" THEN
       "Vuoto"."SetPoint Vuoto Sopra" := "Dati Ciclo"."Passo in Corso"."vuoto sopra";
   END_IF;
   IF #_w1 AND "HMI Ciclo Terminato" THEN "Vuoto"."SetPoint Vuoto Sopra" := 0.0; END_IF;
   #_w2 := "AlwaysTRUE" AND "Manuale";
   IF #_w2 AND "HMI Man Start Vuoto UP" THEN "MK Start Man V UP" := TRUE; END_IF;
   IF #_w2 AND "HMI Man Stop Vuoto UP" THEN
       "HMI Man Start Vuoto UP" := FALSE;
       "MK Start Man V UP" := FALSE;
   END_IF;
   IF #_w2 THEN "Vuoto"."SetPoint Vuoto Sopra" := "Vuoto"."SetPoint Man Vuoto Sopra"; END_IF;
   IF "AlwaysTRUE" AND NOT "Manuale" AND NOT "Automatico Start" THEN "MK Start Man V UP" := FALSE; END_IF;
   "Start Vuoto Sopra" := "AlwaysTRUE" AND ("MK Start Auto V UP" OR "MK Start Man V UP");
   IF "AlwaysTRUE" AND ("Vuoto"."SetPoint Vuoto Sopra" < "Vuoto".K_Altitudine_V_UP) THEN
       "Vuoto"."SetPoint Vuoto Sopra" := "Vuoto".K_Altitudine_V_UP;
   END_IF;
END_REGION

REGION Network 5: Comando Valvole Vuoto
   #_w1 := "AlwaysTRUE" AND "Start Vuoto Sopra";
   "IEC_Timer_0_DB_3".TOF(IN := #_w1 AND ("Vuoto"."Valore Vuoto Sopra" < "Vuoto"."Soglia -2 Grossa Sopra"),
                          PT := T#500MS);
   "MK Ev Vuoto Big Sopra" := "IEC_Timer_0_DB_3".Q;
   "IEC_Timer_0_DB_32".TON(IN := #_w1 AND (("Vuoto"."Valore Vuoto Sopra" < "Vuoto"."Soglia -1 Fine Sopra") OR ("Vuoto"."SetPoint Vuoto Sopra" = 1000.0)),
                           PT := T#500ms);
   "MK Ev Small Vuoto Sopra" := "IEC_Timer_0_DB_32".Q;
END_REGION

REGION Network 6: Comando Valvole aria
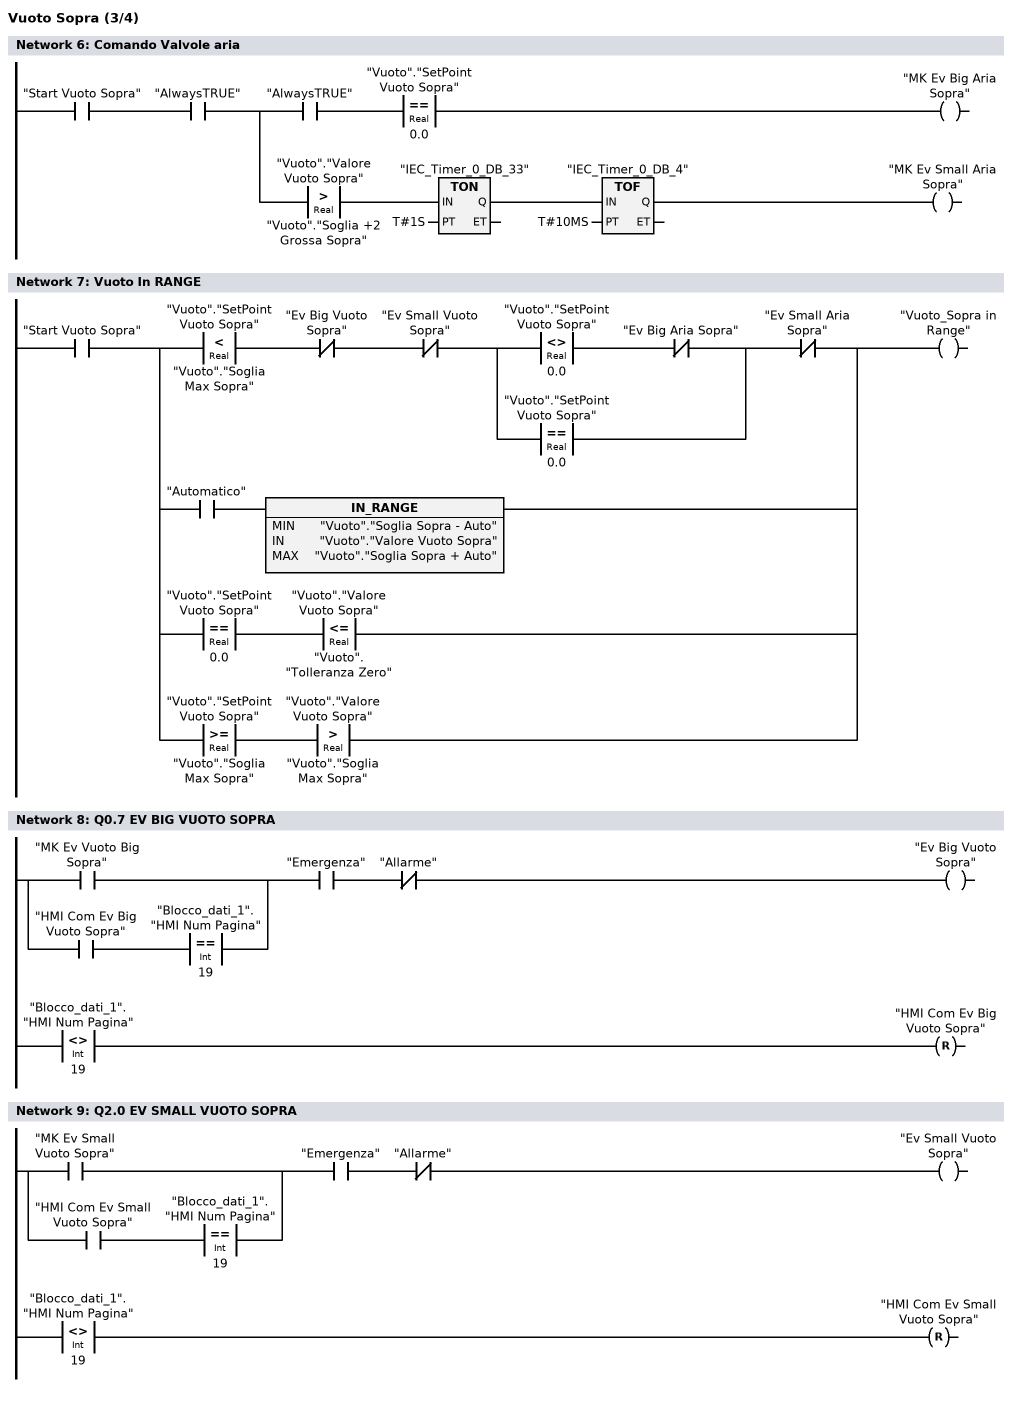
   #_w1 := "Start Vuoto Sopra" AND "AlwaysTRUE";
   "MK Ev Big Aria Sopra" := #_w1 AND "AlwaysTRUE" AND ("Vuoto"."SetPoint Vuoto Sopra" = 0.0);
   "IEC_Timer_0_DB_33".TON(IN := #_w1 AND ("Vuoto"."Valore Vuoto Sopra" > "Vuoto"."Soglia +2 Grossa Sopra"),
                           PT := T#1S);
   "IEC_Timer_0_DB_4".TOF(IN := "IEC_Timer_0_DB_33".Q, PT := T#10MS);
   "MK Ev Small Aria Sopra" := "IEC_Timer_0_DB_4".Q;
END_REGION

REGION Network 7: Vuoto In RANGE
   RUNG wire#powerrail
      Contact( "Start Vuoto Sopra" )
      wire#w1
      { S7_Templates := "SrcType := Real" } LT_Contact(in1 := "Vuoto"."SetPoint Vuoto Sopra", in2 := "Vuoto"."Soglia Max Sopra")
      I_Contact( "Ev Big Vuoto Sopra" )
      I_Contact( "Ev Small Vuoto Sopra" )
      wire#w2
      { S7_Templates := "SrcType := Real" } NE_Contact(in1 := "Vuoto"."SetPoint Vuoto Sopra", in2 := 0.0)
      I_Contact( "Ev Big Aria Sopra" )
      wire#w3
      I_Contact( "Ev Small Aria Sopra" )
      wire#w4
      Coil( "Vuoto_Sopra in Range" )
   END_RUNG
   RUNG wire#w2
      { S7_Templates := "SrcType := Real" } EQ_Contact(in1 := "Vuoto"."SetPoint Vuoto Sopra", in2 := 0.0)
   END_RUNG wire#w3
   RUNG wire#w1
      Contact( "Automatico" )
      { S7_Templates := "SrcType := Real" } InRange(min := "Vuoto"."Soglia Sopra - Auto", in := "Vuoto"."Valore Vuoto Sopra", max := "Vuoto"."Soglia Sopra + Auto")
   END_RUNG wire#w4
   RUNG wire#w1
      { S7_Templates := "SrcType := Real" } EQ_Contact(in1 := "Vuoto"."SetPoint Vuoto Sopra", in2 := 0.0)
      { S7_Templates := "SrcType := Real" } LE_Contact(in1 := "Vuoto"."Valore Vuoto Sopra", in2 := "Vuoto"."Tolleranza Zero")
   END_RUNG wire#w4
   RUNG wire#w1
      { S7_Templates := "SrcType := Real" } GE_Contact(in1 := "Vuoto"."SetPoint Vuoto Sopra", in2 := "Vuoto"."Soglia Max Sopra")
      { S7_Templates := "SrcType := Real" } GT_Contact(in1 := "Vuoto"."Valore Vuoto Sopra", in2 := "Vuoto"."Soglia Max Sopra")
   END_RUNG wire#w4
   // the same network as SCL:
   "Vuoto_Sopra in Range" := "Start Vuoto Sopra" AND ((("Vuoto"."SetPoint Vuoto Sopra" < "Vuoto"."Soglia Max Sopra") AND NOT "Ev Big Vuoto Sopra" AND NOT "Ev Small Vuoto Sopra" AND ((("Vuoto"."SetPoint Vuoto Sopra" <> 0.0) AND NOT "Ev Big Aria Sopra") OR ("Vuoto"."SetPoint Vuoto Sopra" = 0.0)) AND NOT "Ev Small Aria Sopra") OR ("Automatico" AND ("Vuoto"."Soglia Sopra - Auto" <= "Vuoto"."Valore Vuoto Sopra") AND ("Vuoto"."Valore Vuoto Sopra" <= "Vuoto"."Soglia Sopra + Auto")) OR (("Vuoto"."SetPoint Vuoto Sopra" = 0.0) AND ("Vuoto"."Valore Vuoto Sopra" <= "Vuoto"."Tolleranza Zero")) OR (("Vuoto"."SetPoint Vuoto Sopra" >= "Vuoto"."Soglia Max Sopra") AND ("Vuoto"."Valore Vuoto Sopra" > "Vuoto"."Soglia Max Sopra")));
END_REGION

REGION Network 8: Q0.7 EV BIG VUOTO SOPRA
   RUNG wire#powerrail
      Contact( "MK Ev Vuoto Big Sopra" )
      wire#w1
      Contact( "Emergenza" )
      I_Contact( "Allarme" )
      Coil( "Ev Big Vuoto Sopra" )
   END_RUNG
   RUNG wire#powerrail
      Contact( "HMI Com Ev Big Vuoto Sopra" )
      { S7_Templates := "SrcType := Int" } EQ_Contact(in1 := "Blocco_dati_1"."HMI Num Pagina", in2 := 19)
   END_RUNG wire#w1
   RUNG wire#powerrail
      { S7_Templates := "SrcType := Int" } NE_Contact(in1 := "Blocco_dati_1"."HMI Num Pagina", in2 := 19)
      R_Coil( "HMI Com Ev Big Vuoto Sopra" )
   END_RUNG
   // the same network as SCL:
   "Ev Big Vuoto Sopra" := ("MK Ev Vuoto Big Sopra" OR ("HMI Com Ev Big Vuoto Sopra" AND ("Blocco_dati_1"."HMI Num Pagina" = 19))) AND "Emergenza" AND NOT "Allarme";
   IF "Blocco_dati_1"."HMI Num Pagina" <> 19 THEN "HMI Com Ev Big Vuoto Sopra" := FALSE; END_IF;
END_REGION

REGION Network 9: Q2.0 EV SMALL VUOTO SOPRA
   RUNG wire#powerrail
      Contact( "MK Ev Small Vuoto Sopra" )
      wire#w1
      Contact( "Emergenza" )
      I_Contact( "Allarme" )
      Coil( "Ev Small Vuoto Sopra" )
   END_RUNG
   RUNG wire#powerrail
      Contact( "HMI Com Ev Small Vuoto Sopra" )
      { S7_Templates := "SrcType := Int" } EQ_Contact(in1 := "Blocco_dati_1"."HMI Num Pagina", in2 := 19)
   END_RUNG wire#w1
   RUNG wire#powerrail
      { S7_Templates := "SrcType := Int" } NE_Contact(in1 := "Blocco_dati_1"."HMI Num Pagina", in2 := 19)
      R_Coil( "HMI Com Ev Small Vuoto Sopra" )
   END_RUNG
   // the same network as SCL:
   "Ev Small Vuoto Sopra" := ("MK Ev Small Vuoto Sopra" OR ("HMI Com Ev Small Vuoto Sopra" AND ("Blocco_dati_1"."HMI Num Pagina" = 19))) AND "Emergenza" AND NOT "Allarme";
   IF "Blocco_dati_1"."HMI Num Pagina" <> 19 THEN "HMI Com Ev Small Vuoto Sopra" := FALSE; END_IF;
END_REGION

REGION Network 10: Q1.0 EV BIG ARIA SOPRA
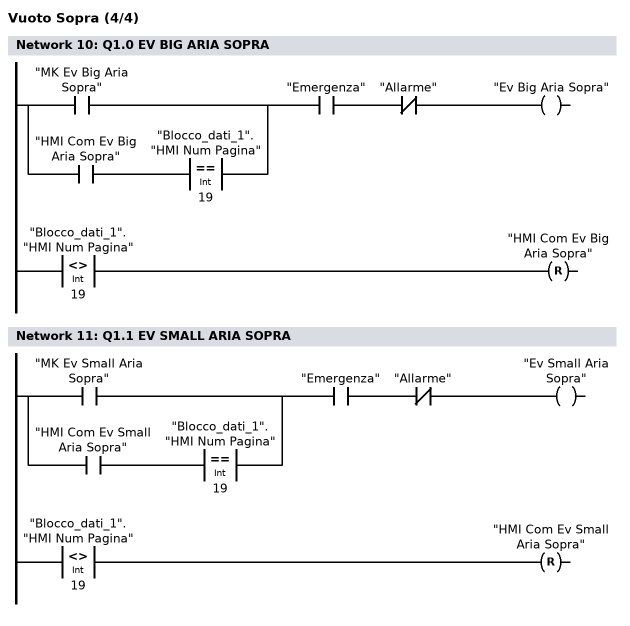
   RUNG wire#powerrail
      Contact( "MK Ev Big Aria Sopra" )
      wire#w1
      Contact( "Emergenza" )
      I_Contact( "Allarme" )
      Coil( "Ev Big Aria Sopra" )
   END_RUNG
   RUNG wire#powerrail
      Contact( "HMI Com Ev Big Aria Sopra" )
      { S7_Templates := "SrcType := Int" } EQ_Contact(in1 := "Blocco_dati_1"."HMI Num Pagina", in2 := 19)
   END_RUNG wire#w1
   RUNG wire#powerrail
      { S7_Templates := "SrcType := Int" } NE_Contact(in1 := "Blocco_dati_1"."HMI Num Pagina", in2 := 19)
      R_Coil( "HMI Com Ev Big Aria Sopra" )
   END_RUNG
   // the same network as SCL:
   "Ev Big Aria Sopra" := ("MK Ev Big Aria Sopra" OR ("HMI Com Ev Big Aria Sopra" AND ("Blocco_dati_1"."HMI Num Pagina" = 19))) AND "Emergenza" AND NOT "Allarme";
   IF "Blocco_dati_1"."HMI Num Pagina" <> 19 THEN "HMI Com Ev Big Aria Sopra" := FALSE; END_IF;
END_REGION

REGION Network 11: Q1.1 EV SMALL ARIA SOPRA
   RUNG wire#powerrail
      Contact( "MK Ev Small Aria Sopra" )
      wire#w1
      Contact( "Emergenza" )
      I_Contact( "Allarme" )
      Coil( "Ev Small Aria Sopra" )
   END_RUNG
   RUNG wire#powerrail
      Contact( "HMI Com Ev Small Aria Sopra" )
      { S7_Templates := "SrcType := Int" } EQ_Contact(in1 := "Blocco_dati_1"."HMI Num Pagina", in2 := 19)
   END_RUNG wire#w1
   RUNG wire#powerrail
      { S7_Templates := "SrcType := Int" } NE_Contact(in1 := "Blocco_dati_1"."HMI Num Pagina", in2 := 19)
      R_Coil( "HMI Com Ev Small Aria Sopra" )
   END_RUNG
   // the same network as SCL:
   "Ev Small Aria Sopra" := ("MK Ev Small Aria Sopra" OR ("HMI Com Ev Small Aria Sopra" AND ("Blocco_dati_1"."HMI Num Pagina" = 19))) AND "Emergenza" AND NOT "Allarme";
   IF "Blocco_dati_1"."HMI Num Pagina" <> 19 THEN "HMI Com Ev Small Aria Sopra" := FALSE; END_IF;
END_REGION
END_FUNCTION

FUNCTION "Pompa Vuoto" : Void   // FC14, LAD
{ S7_Optimized_Access := 'TRUE' }
VERSION : 0.1
   VAR_TEMP   // added for the SCL form of the ladder/FBD networks
      _w1 : Bool;
      _w2 : Bool;
      _w3 : Bool;
      _w4 : Bool;
   END_VAR
BEGIN

REGION Network 1: COMANDO POMPA VUOTO
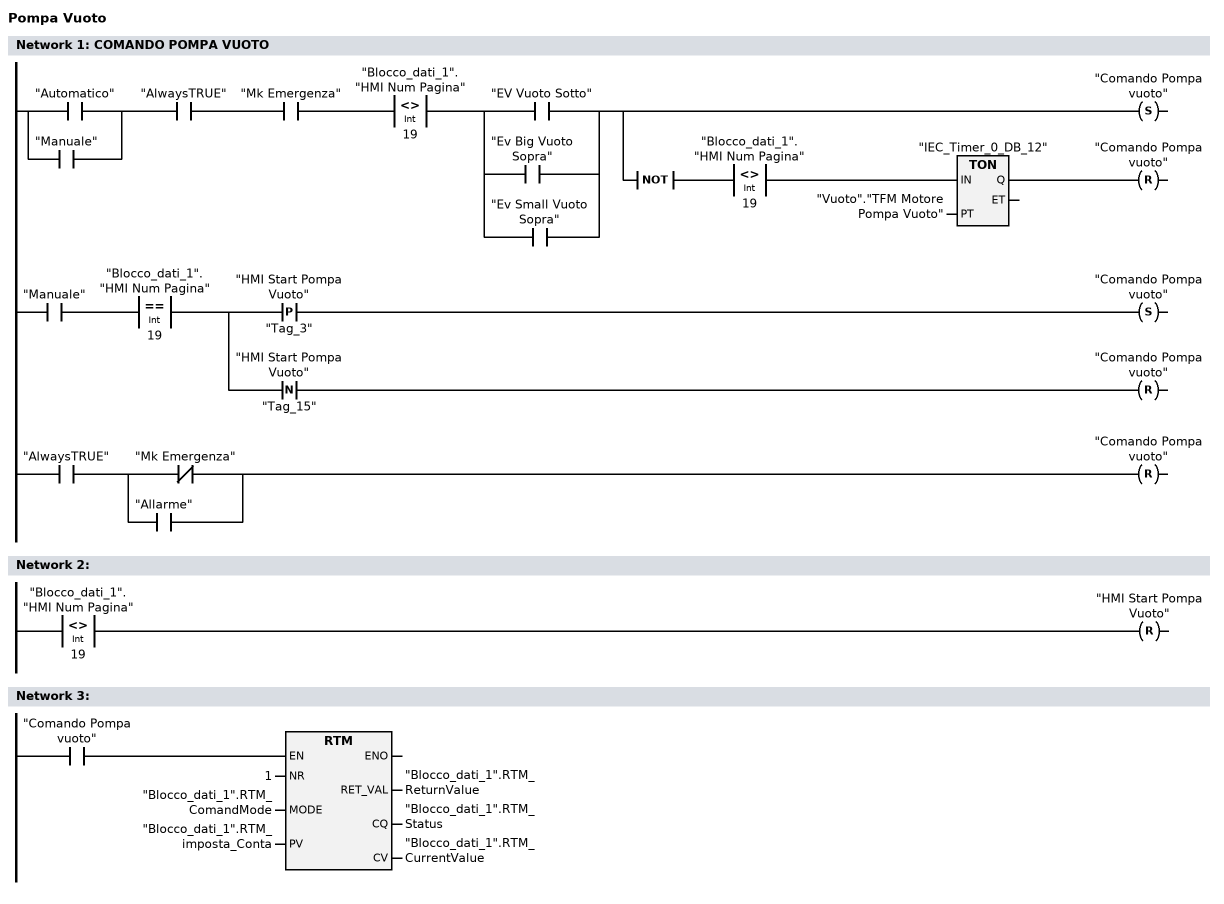
   #_w1 := ("Automatico" OR "Manuale") AND "AlwaysTRUE" AND "Mk Emergenza" AND ("Blocco_dati_1"."HMI Num Pagina" <> 19) AND ("EV Vuoto Sotto" OR "Ev Big Vuoto Sopra" OR "Ev Small Vuoto Sopra");
   IF #_w1 THEN "Comando Pompa vuoto" := TRUE; END_IF;
   "IEC_Timer_0_DB_12".TON(IN := NOT #_w1 AND ("Blocco_dati_1"."HMI Num Pagina" <> 19),
                           PT := "Vuoto"."TFM Motore Pompa Vuoto");
   IF "IEC_Timer_0_DB_12".Q THEN "Comando Pompa vuoto" := FALSE; END_IF;
   #_w2 := "Manuale" AND ("Blocco_dati_1"."HMI Num Pagina" = 19);
   #_w3 := #_w2 AND "HMI Start Pompa Vuoto" AND NOT "Tag_3";   // rising edge of "HMI Start Pompa Vuoto"
   "Tag_3" := "HMI Start Pompa Vuoto";
   IF #_w3 THEN "Comando Pompa vuoto" := TRUE; END_IF;
   #_w4 := #_w2 AND NOT "HMI Start Pompa Vuoto" AND "Tag_15";   // falling edge of "HMI Start Pompa Vuoto"
   "Tag_15" := "HMI Start Pompa Vuoto";
   IF #_w4 THEN "Comando Pompa vuoto" := FALSE; END_IF;
   IF "AlwaysTRUE" AND (NOT "Mk Emergenza" OR "Allarme") THEN "Comando Pompa vuoto" := FALSE; END_IF;
END_REGION

REGION Network 2
   RUNG wire#powerrail
      { S7_Templates := "SrcType := Int" } NE_Contact(in1 := "Blocco_dati_1"."HMI Num Pagina", in2 := 19)
      R_Coil( "HMI Start Pompa Vuoto" )
   END_RUNG
   // the same network as SCL:
   IF "Blocco_dati_1"."HMI Num Pagina" <> 19 THEN "HMI Start Pompa Vuoto" := FALSE; END_IF;
END_REGION

REGION Network 3
   IF "Comando Pompa vuoto" THEN
       "Blocco_dati_1".RTM_ReturnValue := RTM(NR := 1,
                               MODE := "Blocco_dati_1".RTM_ComandMode,
                               PV := "Blocco_dati_1".RTM_imposta_Conta,
                               CQ => "Blocco_dati_1".RTM_Status,
                               CV => "Blocco_dati_1".RTM_CurrentValue);
   END_IF;
END_REGION
END_FUNCTION

FUNCTION "Temperatura Sotto" : Void   // FC15, LAD
{ S7_Optimized_Access := 'TRUE' }
VERSION : 0.1
   VAR_TEMP   // added for the SCL form of the ladder/FBD networks
      _w1 : Bool;
   END_VAR
BEGIN

REGION Network 1
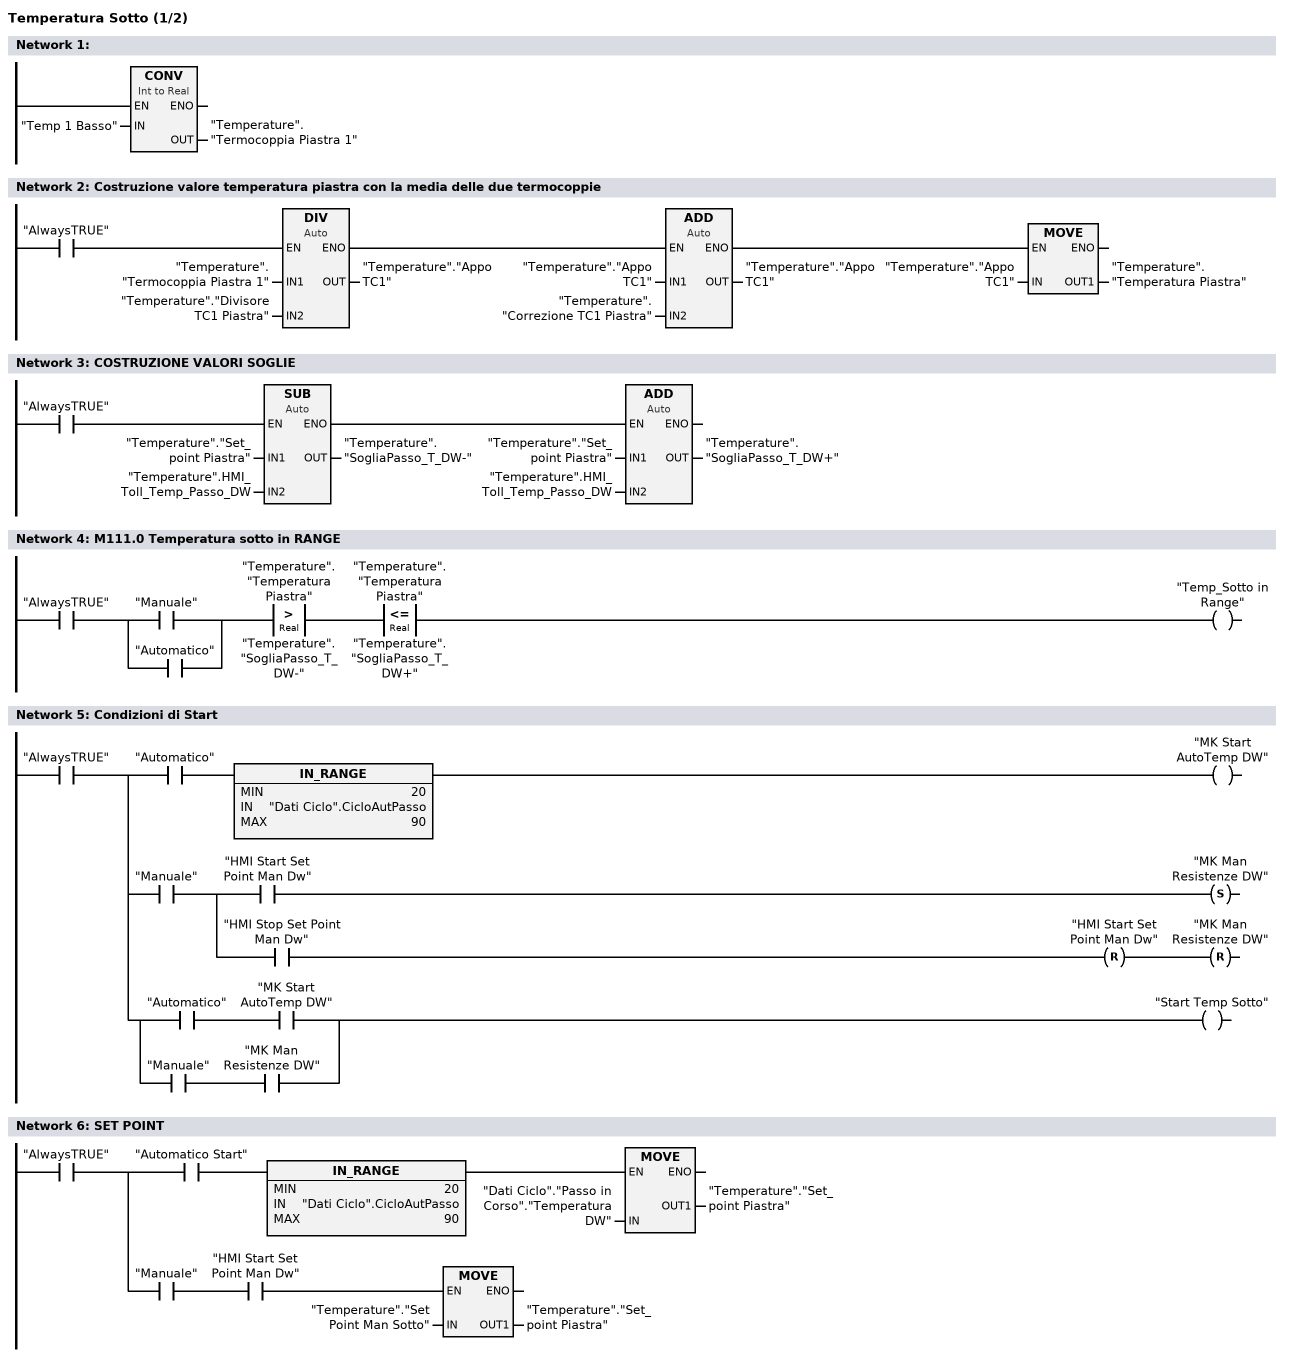
   RUNG wire#powerrail
      { S7_Templates := "[SrcType := Int, DestType := Real]" } Convert(in := "Temp 1 Basso", out => "Temperature"."Termocoppia Piastra 1")
   END_RUNG
   // the same network as SCL:
   "Temperature"."Termocoppia Piastra 1" := INT_TO_REAL("Temp 1 Basso");
END_REGION

REGION Network 2: Costruzione valore temperatura piastra con la media delle due termocoppie
   RUNG wire#powerrail
      Contact( "AlwaysTRUE" )
      Div(in1 := "Temperature"."Termocoppia Piastra 1", in2 := "Temperature"."Divisore TC1 Piastra", out => "Temperature"."Appo TC1")
      Add(in1 := "Temperature"."Appo TC1", in2 := "Temperature"."Correzione TC1 Piastra", out => "Temperature"."Appo TC1")
      Move(in := "Temperature"."Appo TC1", out1 => "Temperature"."Temperatura Piastra")
   END_RUNG
   // the same network as SCL:
   IF "AlwaysTRUE" THEN
       "Temperature"."Appo TC1" := "Temperature"."Termocoppia Piastra 1" / "Temperature"."Divisore TC1 Piastra";
       "Temperature"."Appo TC1" := "Temperature"."Appo TC1" + "Temperature"."Correzione TC1 Piastra";
       "Temperature"."Temperatura Piastra" := "Temperature"."Appo TC1";
   END_IF;
END_REGION

REGION Network 3: COSTRUZIONE VALORI SOGLIE
   RUNG wire#powerrail
      Contact( "AlwaysTRUE" )
      Sub(in1 := "Temperature"."Set_point Piastra", in2 := "Temperature".HMI_Toll_Temp_Passo_DW, out => "Temperature"."SogliaPasso_T_DW-")
      Add(in1 := "Temperature"."Set_point Piastra", in2 := "Temperature".HMI_Toll_Temp_Passo_DW, out => "Temperature"."SogliaPasso_T_DW+")
   END_RUNG
   // the same network as SCL:
   IF "AlwaysTRUE" THEN
       "Temperature"."SogliaPasso_T_DW-" := "Temperature"."Set_point Piastra" - "Temperature".HMI_Toll_Temp_Passo_DW;
       "Temperature"."SogliaPasso_T_DW+" := "Temperature"."Set_point Piastra" + "Temperature".HMI_Toll_Temp_Passo_DW;
   END_IF;
END_REGION

REGION Network 4: M111.0 Temperatura sotto in RANGE
   RUNG wire#powerrail
      Contact( "AlwaysTRUE" )
      wire#w1
      Contact( "Manuale" )
      wire#w2
      { S7_Templates := "SrcType := Real" } GT_Contact(in1 := "Temperature"."Temperatura Piastra", in2 := "Temperature"."SogliaPasso_T_DW-")
      { S7_Templates := "SrcType := Real" } LE_Contact(in1 := "Temperature"."Temperatura Piastra", in2 := "Temperature"."SogliaPasso_T_DW+")
      Coil( "Temp_Sotto in Range" )
   END_RUNG
   RUNG wire#w1
      Contact( "Automatico" )
   END_RUNG wire#w2
   // the same network as SCL:
   "Temp_Sotto in Range" := "AlwaysTRUE" AND ("Manuale" OR "Automatico") AND ("Temperature"."Temperatura Piastra" > "Temperature"."SogliaPasso_T_DW-") AND ("Temperature"."Temperatura Piastra" <= "Temperature"."SogliaPasso_T_DW+");
END_REGION

REGION Network 5: Condizioni di Start
   RUNG wire#powerrail
      Contact( "AlwaysTRUE" )
      wire#w1
      Contact( "Automatico" )
      { S7_Templates := "SrcType := Int" } InRange(min := 20, in := "Dati Ciclo".CicloAutPasso, max := 90)
      Coil( "MK Start AutoTemp DW" )
   END_RUNG
   RUNG wire#w1
      Contact( "Manuale" )
      wire#w2
      Contact( "HMI Start Set Point Man Dw" )
      S_Coil( "MK Man Resistenze DW" )
   END_RUNG
   RUNG wire#w2
      Contact( "HMI Stop Set Point Man Dw" )
      R_Coil( "HMI Start Set Point Man Dw" )
      R_Coil( "MK Man Resistenze DW" )
   END_RUNG
   RUNG wire#w1
      Contact( "Automatico" )
      Contact( "MK Start AutoTemp DW" )
      wire#w3
      Coil( "Start Temp Sotto" )
   END_RUNG
   RUNG wire#w1
      Contact( "Manuale" )
      Contact( "MK Man Resistenze DW" )
   END_RUNG wire#w3
   // the same network as SCL:
   "MK Start AutoTemp DW" := "AlwaysTRUE" AND "Automatico" AND (20 <= "Dati Ciclo".CicloAutPasso) AND ("Dati Ciclo".CicloAutPasso <= 90);
   #_w1 := "AlwaysTRUE" AND "Manuale";
   IF #_w1 AND "HMI Start Set Point Man Dw" THEN "MK Man Resistenze DW" := TRUE; END_IF;
   IF #_w1 AND "HMI Stop Set Point Man Dw" THEN
       "HMI Start Set Point Man Dw" := FALSE;
       "MK Man Resistenze DW" := FALSE;
   END_IF;
   "Start Temp Sotto" := "AlwaysTRUE" AND (("Automatico" AND "MK Start AutoTemp DW") OR ("Manuale" AND "MK Man Resistenze DW"));
END_REGION

REGION Network 6: SET POINT
   RUNG wire#powerrail
      Contact( "AlwaysTRUE" )
      wire#w1
      Contact( "Automatico Start" )
      { S7_Templates := "SrcType := Int" } InRange(min := 20, in := "Dati Ciclo".CicloAutPasso, max := 90)
      Move(in := "Dati Ciclo"."Passo in Corso"."Temperatura DW", out1 => "Temperature"."Set_point Piastra")
   END_RUNG
   RUNG wire#w1
      Contact( "Manuale" )
      Contact( "HMI Start Set Point Man Dw" )
      Move(in := "Temperature"."Set Point Man Sotto", out1 => "Temperature"."Set_point Piastra")
   END_RUNG
   // the same network as SCL:
   IF "AlwaysTRUE" AND "Automatico Start" AND (20 <= "Dati Ciclo".CicloAutPasso) AND ("Dati Ciclo".CicloAutPasso <= 90) THEN
       "Temperature"."Set_point Piastra" := "Dati Ciclo"."Passo in Corso"."Temperatura DW";
   END_IF;
   IF "AlwaysTRUE" AND "Manuale" AND "HMI Start Set Point Man Dw" THEN
       "Temperature"."Set_point Piastra" := "Temperature"."Set Point Man Sotto";
   END_IF;
END_REGION

REGION Network 7: Condizioni di RESET Resistenze
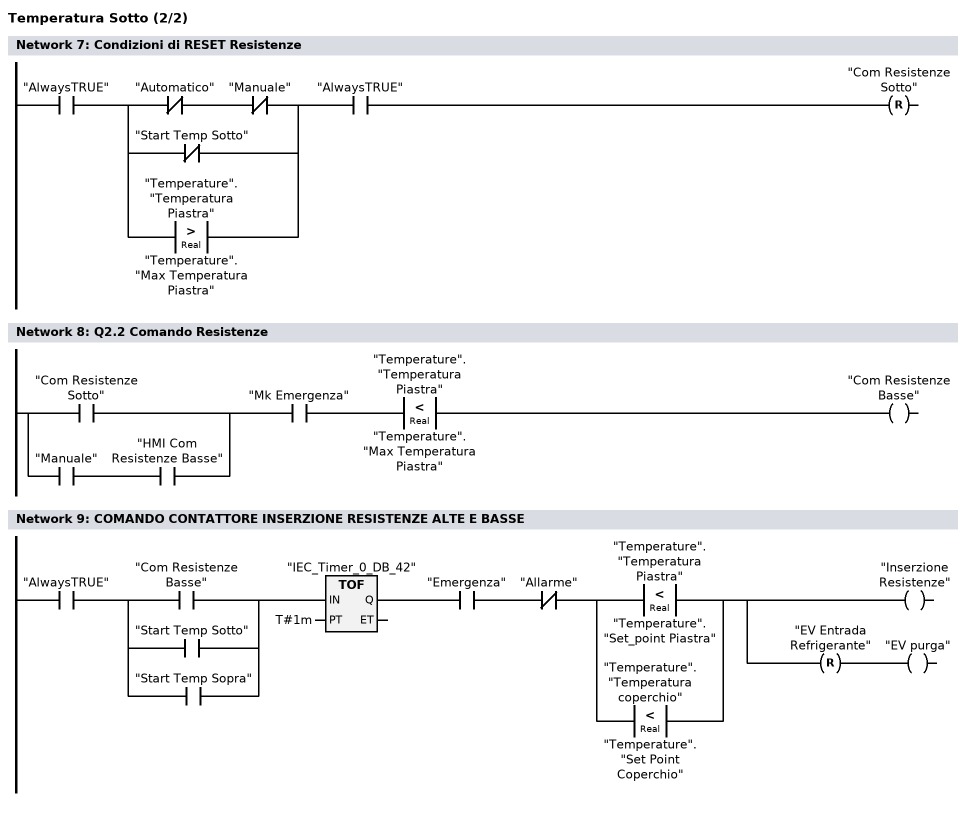
   RUNG wire#powerrail
      Contact( "AlwaysTRUE" )
      wire#w1
      I_Contact( "Automatico" )
      I_Contact( "Manuale" )
      wire#w2
      Contact( "AlwaysTRUE" )
      R_Coil( "Com Resistenze Sotto" )
   END_RUNG
   RUNG wire#w1
      I_Contact( "Start Temp Sotto" )
   END_RUNG wire#w2
   RUNG wire#w1
      { S7_Templates := "SrcType := Real" } GT_Contact(in1 := "Temperature"."Temperatura Piastra", in2 := "Temperature"."Max Temperatura Piastra")
   END_RUNG wire#w2
   // the same network as SCL:
   IF "AlwaysTRUE" AND ((NOT "Automatico" AND NOT "Manuale") OR NOT "Start Temp Sotto" OR ("Temperature"."Temperatura Piastra" > "Temperature"."Max Temperatura Piastra")) AND "AlwaysTRUE" THEN
       "Com Resistenze Sotto" := FALSE;
   END_IF;
END_REGION

REGION Network 8: Q2.2 Comando Resistenze
   RUNG wire#powerrail
      Contact( "Com Resistenze Sotto" )
      wire#w1
      Contact( "Mk Emergenza" )
      { S7_Templates := "SrcType := Real" } LT_Contact(in1 := "Temperature"."Temperatura Piastra", in2 := "Temperature"."Max Temperatura Piastra")
      Coil( "Com Resistenze Basse" )
   END_RUNG
   RUNG wire#powerrail
      Contact( "Manuale" )
      Contact( "HMI Com Resistenze Basse" )
   END_RUNG wire#w1
   // the same network as SCL:
   "Com Resistenze Basse" := ("Com Resistenze Sotto" OR ("Manuale" AND "HMI Com Resistenze Basse")) AND "Mk Emergenza" AND ("Temperature"."Temperatura Piastra" < "Temperature"."Max Temperatura Piastra");
END_REGION

REGION Network 9: COMANDO CONTATTORE INSERZIONE RESISTENZE ALTE E BASSE
   "IEC_Timer_0_DB_42".TOF(IN := "AlwaysTRUE" AND ("Com Resistenze Basse" OR "Start Temp Sotto" OR "Start Temp Sopra"),
                           PT := T#1m);
   "Inserzione Resistenze" := "IEC_Timer_0_DB_42".Q AND "Emergenza" AND NOT "Allarme" AND (("Temperature"."Temperatura Piastra" < "Temperature"."Set_point Piastra") OR ("Temperature"."Temperatura coperchio" < "Temperature"."Set Point Coperchio"));
   IF "Inserzione Resistenze" THEN "EV Entrada Refrigerante" := FALSE; END_IF;
   "EV purga" := "Inserzione Resistenze";
END_REGION
END_FUNCTION

ORGANIZATION_BLOCK "Main"   // OB1, LAD, ProgramCycle
{ S7_Optimized_Access := 'TRUE' }
VERSION : 0.1
   VAR_INPUT
      Initial_Call : Bool;
      Remanence : Bool;
   END_VAR
   VAR_TEMP   // added for the SCL form of the ladder/FBD networks
      _w1 : Bool;
      _w2 : Bool;
      _w3 : Bool;
      _w4 : Bool;
      _w5 : Bool;
   END_VAR
BEGIN

REGION Network 1
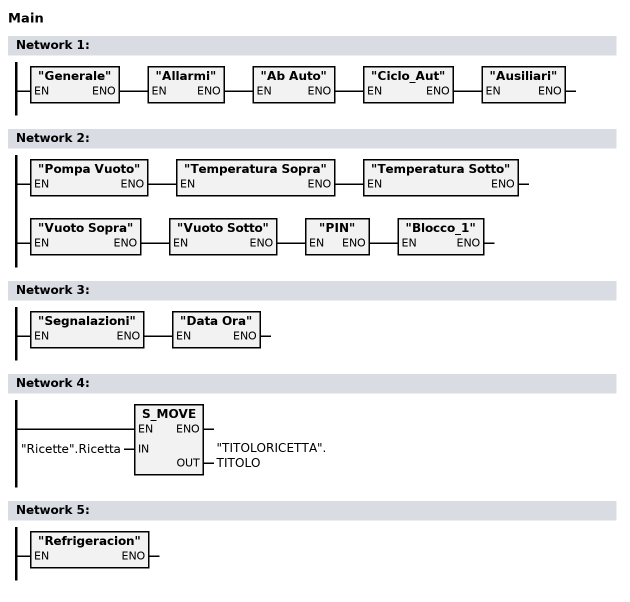
   RUNG wire#powerrail
      "Generale"()
      "Allarmi"()
      "Ab Auto"()
      "Ciclo_Aut"()
      "Ausiliari"()
   END_RUNG
   // the same network as SCL:
   "Generale"(ENO => #_w1);
   "Allarmi"(EN := #_w1, ENO => #_w2);
   "Ab Auto"(EN := #_w2, ENO => #_w3);
   "Ciclo_Aut"(EN := #_w3, ENO => #_w4);
   IF #_w4 THEN "Ausiliari"(); END_IF;
END_REGION

REGION Network 2
   RUNG wire#powerrail
      "Pompa Vuoto"()
      "Temperatura Sopra"()
      "Temperatura Sotto"()
   END_RUNG
   RUNG wire#powerrail
      "Vuoto Sopra"()
      "Vuoto Sotto"()
      "PIN"()
      "Blocco_1"()
   END_RUNG
   // the same network as SCL:
   "Pompa Vuoto"(ENO => #_w1);
   "Temperatura Sopra"(EN := #_w1, ENO => #_w2);
   IF #_w2 THEN "Temperatura Sotto"(); END_IF;
   "Vuoto Sopra"(ENO => #_w3);
   "Vuoto Sotto"(EN := #_w3, ENO => #_w4);
   "PIN"(EN := #_w4, ENO => #_w5);
   IF #_w5 THEN "Blocco_1"(); END_IF;
END_REGION

REGION Network 3
   RUNG wire#powerrail
      "Segnalazioni"()
      "Data Ora"()
   END_RUNG
   // the same network as SCL:
   "Segnalazioni"(ENO => #_w1);
   IF #_w1 THEN "Data Ora"(); END_IF;
END_REGION

REGION Network 4
   RUNG wire#powerrail
      S_Move(in := "Ricette".Ricetta, out => "TITOLORICETTA".TITOLO)
   END_RUNG
   // the same network as SCL:
   "TITOLORICETTA".TITOLO := "Ricette".Ricetta;
END_REGION

REGION Network 5
   RUNG wire#powerrail
      "Refrigeracion"()
   END_RUNG
   // the same network as SCL:
   "Refrigeracion"();
END_REGION
END_ORGANIZATION_BLOCK

ORGANIZATION_BLOCK "Cyclic interrupt"   // OB30, LAD, CyclicInterrupt
{ S7_Optimized_Access := 'TRUE' }
VERSION : 0.1
   VAR_INPUT
      Initial_Call : Bool;   // Initial call of this OB
      Event_Count : Int;   // Events discarded
   END_VAR
BEGIN

REGION Network 1
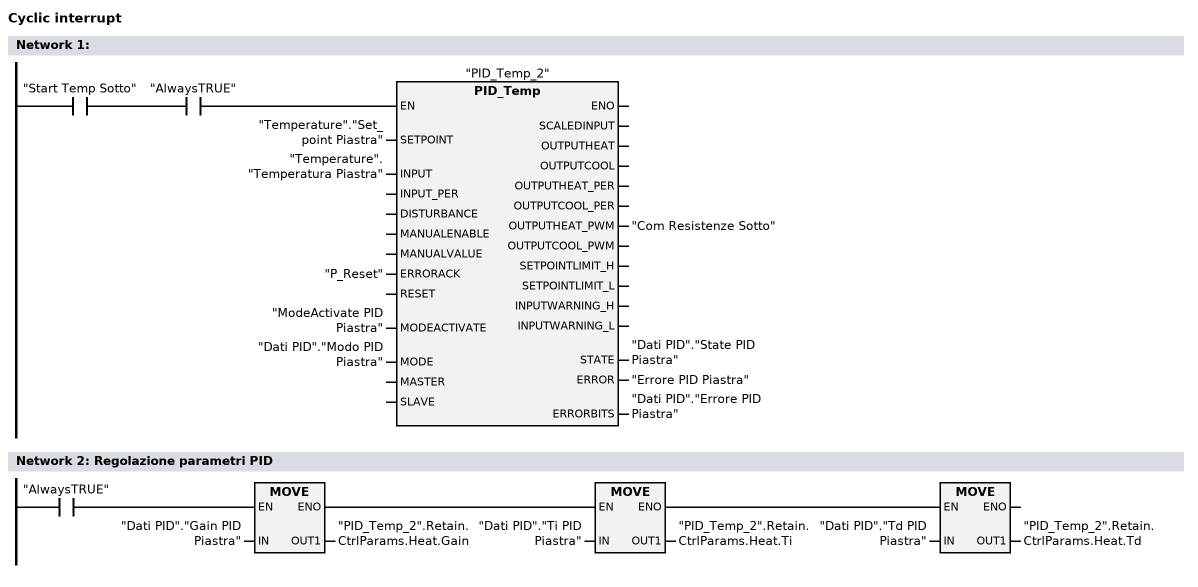
   IF "Start Temp Sotto" AND "AlwaysTRUE" THEN
       "PID_Temp_2"(Setpoint := "Temperature"."Set_point Piastra",   // PID_Temp
                    Input := "Temperature"."Temperatura Piastra",
                    ErrorAck := "P_Reset",
                    ModeActivate := "ModeActivate PID Piastra",
                    Mode := "Dati PID"."Modo PID Piastra",
                    OutputHeat_PWM => "Com Resistenze Sotto",
                    State => "Dati PID"."State PID Piastra",
                    Error => "Errore PID Piastra",
                    ErrorBits => "Dati PID"."Errore PID Piastra");
   END_IF;
END_REGION

REGION Network 2: Regolazione parametri PID
   RUNG wire#powerrail
      Contact( "AlwaysTRUE" )
      Move(in := "Dati PID"."Gain PID Piastra", out1 => "PID_Temp_2".Retain.CtrlParams.Heat.Gain)
      Move(in := "Dati PID"."Ti PID Piastra", out1 => "PID_Temp_2".Retain.CtrlParams.Heat.Ti)
      Move(in := "Dati PID"."Td PID Piastra", out1 => "PID_Temp_2".Retain.CtrlParams.Heat.Td)
   END_RUNG
   // the same network as SCL:
   IF "AlwaysTRUE" THEN
       "PID_Temp_2".Retain.CtrlParams.Heat.Gain := "Dati PID"."Gain PID Piastra";
       "PID_Temp_2".Retain.CtrlParams.Heat.Ti := "Dati PID"."Ti PID Piastra";
       "PID_Temp_2".Retain.CtrlParams.Heat.Td := "Dati PID"."Td PID Piastra";
   END_IF;
END_REGION
END_ORGANIZATION_BLOCK